(* PLC project Система умного дома.project, CODESYS CODESYS V3.5 SP17 Patch 3 *)
(* stored: creationDateTime 2026-04-06T20:38:17.5908527, modificationDateTime 2026-03-25T09:46:39.3897592 *)

{attribute 'qualified_only'}
{attribute 'strict'}
TYPE E_ALERT_PRIORITY : (ALERT_PRIORITY_NONE := 0, ALERT_PRIORITY_LOW := 1, ALERT_PRIORITY_MEDIUM := 2, ALERT_PRIORITY_HIGH := 3, ALERT_PRIORITY_CRITICAL := 4) BYTE;
END_TYPE

{attribute 'qualified_only'}
{attribute 'strict'}
TYPE E_Debug_Log_Level : (LOG_LEVEL_MINIMAL := 0, LOG_LEVEL_NORMAL := 1, LOG_LEVEL_VERBOSE := 2, LOG_LEVEL_DEBUG := 3) BYTE;
END_TYPE

{attribute 'qualified_only'}
{attribute 'strict'}
TYPE E_Lifetime_Device_Type : (LIFETIME_DEVICE_PUMP := 1, LIFETIME_DEVICE_FAN := 2) BYTE;
END_TYPE

{attribute 'qualified_only'}
{attribute 'strict'}
TYPE E_Outdoor_Mode : (OUTDOOR_MODE_AUTO := 0, OUTDOOR_MODE_PARTY := 1, OUTDOOR_MODE_SECURITY := 2, OUTDOOR_MODE_ECONOMY := 3, OUTDOOR_MODE_MANUAL := 4) BYTE;
END_TYPE

{attribute 'qualified_only'}
{attribute 'strict'}
TYPE E_PLC_ROLE : (ROLE_UNDEFINED := 0, ROLE_ACTIVE := 1, ROLE_STANDBY := 2, ROLE_OFFLINE := 3) USINT;
END_TYPE

{attribute 'qualified_only'}
{attribute 'strict'}
TYPE E_Rule_Action_Type : (ACTION_NONE := 0, ACTION_SET_FLOOR_HEATING := 1, ACTION_SET_LIGHTING_BASE := 2, ACTION_SET_LIGHTING_ACCENT := 3, ACTION_SET_SOCKET := 4, ACTION_SET_VENTILATION := 5, ACTION_SET_BLINDS := 6, ACTION_ACTIVATE_SCENARIO := 7, ACTION_TOGGLE_LIGHTING := 8, ACTION_TOGGLE_SOCKET := 9) BYTE;
END_TYPE

{attribute 'qualified_only'}
{attribute 'strict'}
TYPE E_Rule_Comparison : (COMP_NONE := 0, COMP_EQ := 1, COMP_GT := 2, COMP_LT := 3, COMP_GE := 4, COMP_LE := 5, COMP_IN_RANGE := 6, COMP_TRUE := 7, COMP_FALSE := 8) BYTE;
END_TYPE

(* values of E_Rule_Condition_Type: COND_AND: Логическое И (Rule Chaining); COND_OR: Логическое ИЛИ (Rule Chaining) *)

{attribute 'qualified_only'}
{attribute 'strict'}
TYPE E_Rule_Condition_Type : (COND_NONE := 0, COND_AIR_TEMP := 1, COND_FLOOR_TEMP := 2, COND_HUMIDITY := 3, COND_CO2 := 4, COND_METHANE := 5, COND_CO := 6, COND_DOOR_WINDOW := 7, COND_FLOOD := 8, COND_SMOKE := 9, COND_MOTION := 10, COND_TIME_OF_DAY := 11, COND_DAY_OF_WEEK := 12, COND_AND := 13, COND_OR := 14) BYTE;
END_TYPE

{attribute 'qualified_only'}
{attribute 'strict'}
TYPE E_SCENARIO_TYPE : (SCENARIO_NONE := 0, SCENARIO_MORNING := 1, SCENARIO_EVENING := 2, SCENARIO_AWAY := 3, SCENARIO_PARTY := 4, SCENARIO_SLEEP := 5, SCENARIO_EMERGENCY := 6, SCENARIO_PRESENCE := 7) BYTE;
END_TYPE

{attribute 'qualified_only'}
{attribute 'strict'}
TYPE E_SENSOR_TYPE : (SENSOR_TYPE_NONE := 0, SENSOR_TYPE_DOOR_WINDOW := 5, SENSOR_TYPE_GLASS_BREAK := 6, SENSOR_TYPE_FLOOD := 7, SENSOR_TYPE_SMOKE := 8, SENSOR_TYPE_GAS_METHANE := 1, SENSOR_TYPE_GAS_CO := 2, SENSOR_TYPE_TEMP_FLOOR := 3, SENSOR_TYPE_TEMP_AIR := 4) USINT;
END_TYPE

{attribute 'qualified_only'}
{attribute 'strict'}
TYPE E_Trend_Parameter_Type : (TREND_PARAM_NONE := 0, TREND_PARAM_TEMP_AIR := 1, TREND_PARAM_TEMP_FLOOR := 2, TREND_PARAM_PRESSURE := 3, TREND_PARAM_PUMP_CURRENT := 4, TREND_PARAM_GAS_METHANE := 5, TREND_PARAM_GAS_CO := 6) BYTE;
END_TYPE

{attribute 'qualified_only'}
{attribute 'strict'}
TYPE E_TwoFactor_Method : (TF_METHOD_NONE := 0, TF_METHOD_RFID := 1, TF_METHOD_TOTP := 2, TF_METHOD_BOTH := 3) BYTE;
END_TYPE

{attribute 'qualified_only'}
{attribute 'strict'}
TYPE E_Valve_Test_Result : (TEST_RESULT_NONE := 0, TEST_RESULT_PASSED := 1, TEST_RESULT_CURRENT_DEVIATION := 2, TEST_RESULT_TIME_DEVIATION := 3, TEST_RESULT_STALL := 4, TEST_RESULT_LIMIT_SWITCH_FAIL := 5, TEST_RESULT_ABORTED := 6) BYTE;
END_TYPE

(* values of E_VALVE_TYPE: VALVE_NC: Нормально-закрытый; VALVE_NO: Нормально-открытый *)

{attribute 'qualified_only'}
{attribute 'strict'}
TYPE E_VALVE_TYPE : (VALVE_NC := 1, VALVE_NO := 2) USINT;
END_TYPE

{attribute 'qualified_only'}
{attribute 'strict'}
TYPE E_VENTILATION_LOCATION : (VENT_LOCATION_NONE := 0, VENT_LOCATION_BASEMENT_GAME_ROOM := 1, VENT_LOCATION_BASEMENT_GYM := 2, VENT_LOCATION_BASEMENT_BOILER_ROOM := 3, VENT_LOCATION_BATHROOM_1F := 4, VENT_LOCATION_BATHROOM_2F := 5, VENT_LOCATION_MASTER_BATHROOM := 6, VENT_LOCATION_LAUNDRY := 7, VENT_LOCATION_KITCHEN := 8) BYTE;
END_TYPE

{attribute 'qualified_only'}
{attribute 'strict'}
TYPE E_VENTILATION_UNIT_TYPE : (VENTILATION_TYPE_NONE := 0, VENTILATION_TYPE_SUPPLY := 1, VENTILATION_TYPE_EXHAUST := 2) USINT;
END_TYPE

{attribute 'qualified_only'}
{attribute 'strict'}
TYPE E_WEATHER_COMPENSATION_METHOD : (WEATHER_COMP_NONE := 0, WEATHER_COMP_OUTDOOR_RESET := 1) USINT;
END_TYPE

{attribute 'qualified_only'}
{attribute 'strict'}
TYPE E_Zone_Access_Level : (ZONE_ACCESS_NONE := 0, ZONE_ACCESS_VIEW := 1, ZONE_ACCESS_CONTROL := 2, ZONE_ACCESS_CONFIG := 3, ZONE_ACCESS_FULL := 4) BYTE;
END_TYPE

TYPE ST_Astro_Time : STRUCT
  sunrise_ms : UDINT := 0;
  sunset_ms : UDINT := 0;
  is_daylight : BOOL := FALSE;
END_STRUCT;
END_TYPE

TYPE ST_BlackBox_Record : STRUCT
  Timestamp : UDINT;
  Gas_Methane_LEL : REAL;
  Gas_CO_PPM : REAL;
  Flood_Active : BOOL;
  Fire_Active : BOOL;
  Valve_Gas_Status : BYTE;
  Valve_Water_Status : BYTE;
  PLC_Active_ID : BYTE;
END_STRUCT;
END_TYPE

TYPE ST_Boiler_Status : STRUCT
  Active : BOOL;
  Running : BOOL;
  Error : BOOL;
  Power_Percent : REAL;
  Current_Power : REAL;
  Work_Seconds : UDINT;
  Work_Hours : REAL;
  Resource_Percent : REAL := 100;
  Last_Start : DT;
END_STRUCT;
END_TYPE

TYPE ST_Component_Maintenance : STRUCT
  Is_Faulty : BOOL;  (* Устройство неисправно *)
  Is_In_Maintenance : BOOL;  (* Выведено в ремонт вручную *)
  Fallback_Value : REAL;  (* Значение для подстановки (0-100% или температура) *)
  Use_Last_Good_Value : BOOL;  (* Использовать последнее достоверное значение *)
END_STRUCT;
END_TYPE

TYPE ST_Debug_Log_Record : STRUCT
  timestamp_ms : UDINT;
  level : BYTE;  (* E_Debug_Log_Level *)
  source_id : BYTE;
  event_code : WORD;
  value_int : UDINT;
  value_real : REAL;
  text : STRING(80);
  crc32 : DWORD;
END_STRUCT;
END_TYPE

TYPE ST_Debug_Logger_Config : STRUCT
  enabled : BOOL;
  sampling_period_ms : UDINT := 1000;
END_STRUCT;
END_TYPE

TYPE ST_Device_Health : STRUCT
  Health_Score : BYTE := 100;  (* 0..100% *)
  Total_Runtime_Hours : UDINT;
  Starts_Count : UDINT;
  Last_Start_Current : REAL;
  Avg_Start_Current : REAL;
  Maintenance_Required : BOOL;
  Warning_Message : STRING(50);
END_STRUCT;
END_TYPE

TYPE ST_DHW_Config : STRUCT
  Target_Temp : REAL := 55;
  Hysteresis : REAL := 2;
  Circulation_Schedule_Enabled : BOOL := TRUE;
  Circulation_Start : TOD := TIME_OF_DAY#6:0;
  Circulation_End : TOD := TIME_OF_DAY#23:0;
  Anti_Legionella_Enabled : BOOL := TRUE;
  Anti_Legionella_Day : UINT := 7;  (* Воскресенье *)
END_STRUCT;
END_TYPE

TYPE ST_DHW_Status : STRUCT
  Temp : REAL;
  Pressure : REAL;
  Heating_Pump_On : BOOL;
  Circ_Pump_On : BOOL;
  Error : BOOL;
  Error_ID : WORD;
END_STRUCT;
END_TYPE

TYPE ST_Flood_Config : STRUCT
  Emergency_Two_Stage_Enabled : BOOL := TRUE;  (* ТЗ 4.4 *)
  Valve_Test_Period_Days : UINT := 7;  (* ТЗ 12.2 *)
  Current_Threshold_MA : REAL := 500;  (* Порог тока для диагностики *)
END_STRUCT;
END_TYPE

TYPE ST_Flood_Global_Config : STRUCT
  valve_types : ARRAY[1..3] OF E_VALVE_TYPE := [3(E_VALVE_TYPE.VALVE_NC)];
  min_duration_ms : UDINT := 30000;
END_STRUCT;
END_TYPE

TYPE ST_FloorHeating_Circuit_Config : STRUCT
  circuit_id : BYTE := 0;
  zone : BYTE := 0;
  design_temp : REAL := 35;
  min_temp : REAL := 20;
  max_temp : REAL := 45;
  pid_kp : REAL := 2;
END_STRUCT;
END_TYPE

TYPE ST_FloorHeating_Global_Config : STRUCT
  enable_floor_heating : BOOL := TRUE;
  anti_freeze_temp : REAL := 7;
  overheat_temp : REAL := 45;
  weather_compensation_enabled : BOOL := TRUE;
  total_circuits : BYTE := 16;
END_STRUCT;
END_TYPE

TYPE ST_FloorHeating_Manifold_Config : STRUCT
  manifold_id : BYTE;
  location : STRING(30);
  nominal_flow : REAL;
  enable_pump : BOOL;
  circuits : ARRAY[1..4] OF ST_FloorHeating_Circuit_Config;
END_STRUCT;
END_TYPE

TYPE ST_Gas_Valve_Configuration : STRUCT
  valve_id : BYTE := 0;
  valve_type : E_VALVE_TYPE := E_VALVE_TYPE.VALVE_NC;
  close_time_seconds : UDINT := 10;
  open_time_seconds : UDINT := 10;
  emergency_open_allowed : BOOL := FALSE;
END_STRUCT;
END_TYPE

TYPE ST_Gateway_Command : STRUCT
  command_id : UDINT;
  timestamp_ms : UDINT;
  operator_id : STRING(10);
  command_type : BYTE;
  target_zone : BYTE;
  target_value : REAL;
  target_on_off : BOOL;
  target_scenario : E_SCENARIO_TYPE;
  target_armed : BOOL;
  crc32 : DWORD;
END_STRUCT;
END_TYPE

TYPE ST_Heating_Config : STRUCT
  Weather_Comp_Enabled : BOOL := TRUE;
  Weather_Coef : REAL := 0.1;
  Freeze_Threshold : REAL := 7;
  Overheat_Threshold : REAL := 45;
  Night_Reduction : REAL := 3;
  Target_Floor_Temp : REAL := 28;
  Target_Room_Temp : REAL := 22;
  Hysteresis : REAL := 0.5;
END_STRUCT;
END_TYPE

TYPE ST_History_Record : STRUCT
  timestamp_ms : UDINT := 0;
  event_code : WORD := 0;
  event_value : REAL := 0;
  unit : BYTE := 0;
  zone_id : BYTE := 0;
  operator_id : STRING(10) := '';
  priority : E_ALERT_PRIORITY := E_ALERT_PRIORITY.ALERT_PRIORITY_NONE;
END_STRUCT;
END_TYPE

TYPE ST_Lifetime_Status : STRUCT
  device_id : BYTE;
  runtime_hours : UDINT;
  start_count : UDINT;
  remaining_hours : UDINT;
  remaining_percent : BYTE;
  maintenance_required : BOOL;
  last_calc_timestamp : UDINT;
END_STRUCT;
END_TYPE

TYPE ST_Maintenance_Access_Config : STRUCT
  maintenance_enabled : BOOL := FALSE;
  max_duration_minutes : UDINT := 60;
  requires_two_person : BOOL := TRUE;
  access_level_required : BYTE := 2;
END_STRUCT;
END_TYPE

TYPE ST_Manifold_Status : STRUCT
  Pump_On : BOOL;
  Pump_Current : REAL;
  Pressure : REAL;
  Temp_Supply : REAL;
  Temp_Return : REAL;
  Valve_Pos : REAL;  (* 0-100% *)
  Error : BOOL;
  Error_ID : WORD;
END_STRUCT;
END_TYPE

TYPE ST_Operator_Zone_Rights : STRUCT
  operator_id : STRING(10);
  global_access_level : BYTE := 0;
  zone_masks : ARRAY[1..18] OF DWORD;
  last_modified : UDINT;
END_STRUCT;
END_TYPE

TYPE ST_Outdoor_Zone_Config : STRUCT
  zone_id : BYTE := 0;
  lighting_circuit_id : BYTE := 0;
  auto_enabled : BOOL := TRUE;
  party_mode_enabled : BOOL := FALSE;
END_STRUCT;
END_TYPE

TYPE ST_Owen_Analog_Value : STRUCT
  rValue : REAL;  (* Измеренное значение *)
  uiCycleTime : UINT;  (* Циклическое время *)
  wStatus : WORD;  (* Код статуса (ANALOG_SENSOR_ERRORS) *)
END_STRUCT;
END_TYPE

TYPE ST_Rule_Action : STRUCT
  Active : BOOL;
  Target_ID : BYTE;
  Value : REAL;
END_STRUCT;
END_TYPE

TYPE ST_Scenario_Config : STRUCT
  scenario_id : E_SCENARIO_TYPE;
  lighting_level_base : BYTE := 100;
  lighting_level_accent : BYTE := 100;
  floor_heating_adjust_celsius : REAL := 0;
  ventilation_speed_percent : BYTE := 50;
  sockets_enabled : BOOL := TRUE;
  blinds_position_percent : BYTE := 0;
END_STRUCT;
END_TYPE

TYPE ST_Scenario_Transition_Config : STRUCT
  current_scenario : E_SCENARIO_TYPE;
  target_scenario : E_SCENARIO_TYPE;
  min_duration_minutes : UDINT := 5;
  transition_allowed : BOOL := FALSE;
END_STRUCT;
END_TYPE

TYPE ST_Security_Config : STRUCT
  PIN_Code : STRING(4) := '1234';
  Max_Attempts : UINT := 3;
  Entry_Delay_S : UINT := 45;
  Two_Factor_Enabled : BOOL := FALSE;
  Two_Stage_Mode : BOOL := TRUE;  (* ТЗ 3.4 *)
  Confirmation_Timeout_S : UINT := 120;  (* ТЗ 3.4 (60-300с) *)
  Phones : ARRAY[1..5] OF STRING(15);
  gate_open_pulse_ms : UDINT := 1000;  (* Управление доступом *)
  wicket_open_pulse_ms : UDINT := 1000;
  lock_open_pulse_ms : UDINT := 1000;
  lock_close_pulse_ms : UDINT := 1000;
END_STRUCT;
END_TYPE

TYPE ST_Security_Global_Config : STRUCT
  entry_delay_seconds : UDINT := 30;
  exit_delay_seconds : UDINT := 60;
  alarm_duration_seconds : UDINT := 180;
  two_person_timeout_seconds : UDINT := 120;
  max_access_attempts : BYTE := 3;
  auto_arm_enabled : BOOL := FALSE;
  auto_arm_time_ms : UDINT := 0;
  gate_open_pulse_ms : UDINT := 1000;  (* ТЗ: Управление доступом *)
  wicket_open_pulse_ms : UDINT := 1000;
  lock_open_pulse_ms : UDINT := 1000;
  lock_close_pulse_ms : UDINT := 1000;
END_STRUCT;
END_TYPE

TYPE ST_Security_Zone_State : STRUCT
  Armed : BOOL;
  Alarm : BOOL;
  Bypassed : BOOL;
  Last_Trigger_Time : DT;
  Trigger_Count : UINT;
END_STRUCT;
END_TYPE

TYPE ST_Sensor_Calibration_Record : STRUCT
  sensor_id : UDINT := 0;
  sensor_type : E_SENSOR_TYPE;
  zone_id : BYTE := 0;
  offset : REAL := 0;
  multiplier : REAL := 1;
  last_calibration_timestamp : UDINT := 0;
  verification_passed : BOOL := FALSE;
END_STRUCT;
END_TYPE

TYPE ST_State_Snapshot : STRUCT
  timestamp_ms : UDINT := 0;
  operator_id : STRING(10) := '';
  scenario_id : E_SCENARIO_TYPE := E_SCENARIO_TYPE.SCENARIO_NONE;
  lighting_levels : ARRAY[1..16] OF BYTE;
  floor_heating_setpoints : ARRAY[1..16] OF REAL;
  alarm_active : BOOL := FALSE;
  crc32 : DWORD := 0;
END_STRUCT;
END_TYPE

TYPE ST_System_State_Summary : STRUCT
  Outdoor_Temp : REAL;
  Indoor_Temp : ARRAY[1..16] OF REAL;
  Floor_Temps : ARRAY[1..16] OF REAL;
  Humidity : ARRAY[1..8] OF REAL;
  CO2 : ARRAY[1..8] OF REAL;
  Gas_Alarm : BOOL;
  Flood_Alarm : BOOL;
  Fire_Alarm : BOOL;
  Security_Armed : BOOL;
END_STRUCT;
END_TYPE

TYPE ST_Tariff_Config : STRUCT
  Enabled : BOOL := FALSE;
  Night_Start_Hour : UINT := 23;  (* 23:00 *)
  Night_End_Hour : UINT := 7;  (* 07:00 *)
  Boost_Delta : REAL := 2;  (* На сколько градусов поднять уставку ночью *)
END_STRUCT;
END_TYPE

TYPE ST_Trend_Config : STRUCT
  param_type : BYTE;  (* E_Trend_Parameter_Type *)
  zone_id : BYTE;
  enabled : BOOL;
  deviation_threshold_percent : REAL := 10;
  history_days : UDINT := 7;
END_STRUCT;
END_TYPE

TYPE ST_Trend_Data : STRUCT
  config : ST_Trend_Config;
  record_count : UDINT;
  write_index : UDINT;
  sum_values : REAL;
  crc32 : DWORD;
END_STRUCT;
END_TYPE

TYPE ST_Trend_Header : STRUCT
  parameter_type : BYTE;  (* E_Trend_Parameter_Type *)
  zone_id : BYTE := 0;
  records_count : UDINT := 0;
  average_value : REAL := 0;
  min_value : REAL := 0;
  max_value : REAL := 0;
END_STRUCT;
END_TYPE

TYPE ST_Trend_History_Record : STRUCT
  timestamp_ms : UDINT := 0;
  value : REAL := 0;
END_STRUCT;
END_TYPE

TYPE ST_TwoFactor_Auth_State : STRUCT
  operator_id : STRING(10);
  is_pending : BOOL;  (* Ожидание ввода 2-го фактора *)
  start_time : UDINT;
  timeout_ms : UDINT := 60000;
END_STRUCT;
END_TYPE

TYPE ST_TwoFactor_Data : STRUCT
  operator_id : STRING(10);
  AuthMethod : BYTE;  (* E_TwoFactor_Method *)
  rfid_tag : STRING(20);
  totp_secret : STRING(32);
  last_modified : UDINT;
END_STRUCT;
END_TYPE

TYPE ST_User_Rule : STRUCT
  Enabled : BOOL;
  Condition_Type : BYTE;  (* 1-Temp, 2-Hum, 3-CO2, 4-Security, 5-Time *)
  Condition_Op : BYTE;  (* 1:>, 2:<, 3:= *)
  Condition_Value : REAL;
  Action_Target_ID : BYTE;
  Action_Value : REAL;
  Action_Type : BYTE;  (* 1-SetTemp, 2-Switch, 3-Scenario *)
  Priority : BYTE;  (* ТЗ 7.4: Приоритет (0-255) *)
END_STRUCT;
END_TYPE

TYPE ST_Valve_Test_Config : STRUCT
  valve_id : BYTE := 0;
  test_interval_days : UDINT := 7;
  nominal_current_a : REAL := 0.5;
  Nominal_Current : REAL := 0.5;
  nominal_close_time_sec : REAL := 10;
  enabled : BOOL := TRUE;
END_STRUCT;
END_TYPE

TYPE ST_Ventilation_Config : STRUCT
  CO2_Threshold : REAL := 800;
  Humidity_Threshold : REAL := 65;
  Night_Mode_Start : TOD := TIME_OF_DAY#23:0;
  Night_Mode_End : TOD := TIME_OF_DAY#7:0;
END_STRUCT;
END_TYPE

TYPE ST_Ventilation_Global_Config : STRUCT
  enable_ventilation : BOOL := TRUE;
  total_units : BYTE := 8;
  default_supply_speed : BYTE := 40;
  default_exhaust_speed : BYTE := 40;
END_STRUCT;
END_TYPE

TYPE ST_Ventilation_Scenario_Mode : STRUCT
  Scenario_ID : BYTE;
  Scenario_Priority : BYTE;
  Fire_Alarm : BOOL;
  Methane_Alarm : BOOL;
  Smoke_Detected : BOOL;
  Exhaust_Modes : ARRAY[1..5] OF BYTE;
  Supply_Modes : ARRAY[1..3] OF BYTE;
END_STRUCT;
END_TYPE

TYPE ST_Ventilation_Unit : STRUCT
  Enabled : BOOL;
  Speed_Percent : REAL;
  Filter_Dirty : BOOL;
  Error : BOOL;
  Mode : BYTE;  (* 0-Eco, 1-Std, 2-Int, 3-Emergency *)
END_STRUCT;
END_TYPE

TYPE ST_Ventilation_Unit_Config : STRUCT
  unit_id : BYTE := 0;
  unit_type : E_VENTILATION_UNIT_TYPE;
  location : E_VENTILATION_LOCATION;
  min_speed : BYTE := 20;
  max_speed : BYTE := 100;
  Threshold_Hum : REAL := 65;
  has_smoke_detector : BOOL := FALSE;
END_STRUCT;
END_TYPE

TYPE ST_Zone_Sensors : STRUCT
  Temp_Room : REAL;
  Temp_Floor : REAL;
  Motion_Active : BOOL;
  Switch_Physical : BOOL;
  Light_State : BOOL;
  Maintenance : ST_Component_Maintenance;
END_STRUCT;
END_TYPE

{attribute 'qualified_only'}
VAR_GLOBAL  (* GVL_BlackBox *)
  G_BlackBox_Buffer : ARRAY[0..99] OF ST_BlackBox_Record;  (* Буфер на 100 записей (при опросе 100мс это 10 секунд истории) *)
  G_BlackBox_Frozen : BOOL;
  G_BlackBox_LastIndex : INT;
END_VAR

{attribute 'qualified_only'}
VAR_GLOBAL CONSTANT  (* GVL_Constants *)
  C_MS_PER_SEC : UDINT := 1000;
  C_SEC_PER_MIN : UDINT := 60;
  C_MIN_PER_HOUR : UDINT := 60;
  C_MS_PER_MIN : UDINT := 60000;
  C_MAX_RULES : INT := 20;
  C_ZONE_COUNT : BYTE := 18;
END_VAR

{attribute 'qualified_only'}
VAR_GLOBAL  (* GVL_Diagnostics *)
  G_Pump_Health : ARRAY[1..5] OF ST_Device_Health;  (* Для 5 коллекторных насосов *)
  G_Gas_Valve_Health : ST_Device_Health;
  G_System_Health_Summary : BYTE := 100;
END_VAR

{attribute 'qualified_only'}
VAR_GLOBAL  (* GVL_Global_Variables *)
  GVL_System_Time_MS : UDINT;
  GVL_IsActivePLC : BOOL := TRUE;
  GVL_Local_PLC_Role : E_PLC_ROLE := E_PLC_ROLE.ROLE_ACTIVE;
  GVL_Floor_Temps : ARRAY[1..16] OF REAL;  (* Данные датчиков *)
  GVL_Valve_States : ARRAY[1..3] OF BYTE;
END_VAR

VAR_GLOBAL  (* GVL_HMI_Config *)
  G_HMI_FloorHeating_Configs : ARRAY[1..16] OF ST_FloorHeating_Circuit_Config;  (* Настройки отопления (16 контуров) *)
  G_HMI_Tariff_Settings : ST_Tariff_Config;
  G_HMI_Vent_Global_Config : ST_Ventilation_Global_Config;  (* Настройки вентиляции (8 установок) *)
  G_HMI_Vent_Unit_Configs : ARRAY[1..8] OF ST_Ventilation_Unit_Config;
  G_HMI_Scenario_Configs : ARRAY[1..6] OF ST_Scenario_Config;  (* Для каждого типа сценария *)
  G_HMI_Outdoor_Configs : ARRAY[1..4] OF ST_Outdoor_Zone_Config;
  G_HMI_Flood_Config : ST_Flood_Global_Config;  (* Настройки безопасности *)
  G_HMI_Cleaning_Mode_Active : ARRAY[1..3] OF BOOL;  (* Режим уборки для 3-х зон протечки *)
  G_HMI_Cleaning_Mode_TimeLeft : ARRAY[1..3] OF UINT;  (* Оставшееся время (мин) *)
  G_HMI_Gas_Config : ST_Gas_Valve_Configuration;
  G_HMI_Admin_2FA_Enabled : BOOL := FALSE;  (* Настройка: 1 или 2 фактора для ADMIN *)
  G_HMI_Current_Operator_Factor2_Done : BOOL;  (* Флаг прохождения 2-го фактора *)
  G_HMI_Sensor_Calibrations : ARRAY[1..20] OF ST_Sensor_Calibration_Record;  (* Калибровка датчиков (например, для 20 датчиков) *)
  G_HMI_Current_Operator_ID : STRING(10);  (* ID текущего авторизованного пользователя *)
  G_HMI_Manual_Gas_Valve_Open : BOOL;  (* Запрос на открытие *)
  G_HMI_Manual_Gas_Valve_Time : UDINT := 5;  (* Время в минутах *)
  G_HMI_Manual_Gas_Valve_TimeLeft : UDINT;  (* Оставшееся время (для вывода на HMI) *)
  G_HMI_Apply_Settings : BOOL;  (* Команда на сохранение настроек в NVRAM *)
  G_HMI_Gate_Open_Req : BOOL;  (* Управление доступом (HMI) *)
  G_HMI_Wicket_Open_Req : BOOL;
  G_HMI_Lock_1_Open_Req : BOOL;
  G_HMI_Lock_1_Close_Req : BOOL;
  G_HMI_Lock_2_Open_Req : BOOL;
  G_HMI_Lock_2_Close_Req : BOOL;
END_VAR

VAR_GLOBAL  (* GVL_IO *)
  DI_Security_Open : ARRAY[1..15] OF BOOL;  (* Датчики открытия (15 физических каналов по ТЗ 3.1) *)
  DI_Security_Glass : ARRAY[1..15] OF BOOL;  (* Датчики разбития (15 физических каналов по ТЗ 3.2) *)
  DI_Security_2F_Group : BOOL;  (* Групповой канал 2-го этажа *)
  DI_Flood_Sensors : ARRAY[1..12] OF BOOL;  (* Датчики протечки (12 штук по ТЗ 4.1) *)
  AO_Manifold_Valves : ARRAY[1..5] OF UINT;  (* 0-1000 (Modbus) *)
  DO_Manifold_Pumps : ARRAY[1..5] OF BOOL;
  AI_Manifold_Currents : ARRAY[1..5] OF INT;  (* 4-20mA -> 400-2000 *)
  AI_Manifold_Pressures : ARRAY[1..5] OF INT;  (* 0-10V -> 0-1000 *)
  AI_Manifold_Temps_Supply : ARRAY[1..5] OF ST_Owen_Analog_Value;
  AI_Manifold_Temps_Return : ARRAY[1..5] OF INT;
  AO_Supply_Fans : ARRAY[1..3] OF UINT;  (* 0-1000 *)
  AO_Exhaust_Fans : ARRAY[1..5] OF UINT;  (* 0-1000 *)
  DO_Boiler_Enable : ARRAY[1..2] OF BOOL;  (* Котлы (BAXI Luna Platinum+ через OpenTherm) *)
  AO_Boiler_Setpoint : ARRAY[1..2] OF UINT;  (* 0-1000 (0-100.0 C) *)
  AI_Boiler_Modulation : ARRAY[1..2] OF INT;
  AI_Boiler_Flame_Status : ARRAY[1..2] OF BOOL;
  DI_Boiler_Error : ARRAY[1..2] OF BOOL;
  AI_Methane_LEL : ARRAY[1..2] OF ST_Owen_Analog_Value;  (* 0-100% LEL *)
  AI_CO_PPM : ARRAY[1..8] OF REAL;  (* 0-1000 PPM *)
  DI_Smoke_Sensors : ARRAY[1..6] OF BOOL;
  AI_Temp_Outdoor : ST_Owen_Analog_Value;  (* Аналоговые входы (AI) *)
  AI_Floor_Temps : ARRAY[1..16] OF REAL;
  AI_Room_Temps : ARRAY[1..16] OF REAL;  (* Датчики температуры помещения (ТЗ 1.1) *)
  DO_Zone_Valves : ARRAY[1..16] OF BOOL;  (* Клапаны контуров ТП *)
  AI_DHW_Temp : REAL;  (* ГВС (ТЗ 5.0) *)
  AI_DHW_Pressure : REAL;
  DO_DHW_Heating_Pump : BOOL;
  DO_DHW_Circ_Pump : BOOL;
  DI_Lighting_Switches : ARRAY[1..16] OF BOOL;  (* Освещение и Движение (ТЗ 1.0, 2.0) *)
  DI_Motion_Sensors : ARRAY[1..16] OF BOOL;
  DO_Gas_Valve_Close : BOOL;  (* Безопасность и Аварии *)
  DO_Water_Valve_35_Close : BOOL;
  DO_Water_Valve_36_Close : BOOL;
  AI_Water_Valve_35_Current : REAL;
  AI_Water_Valve_36_Current : REAL;
  DI_Power_OK : BOOL;
  DO_Gas_Siren : BOOL;
  DO_Fire_Siren : BOOL;
  DO_Pump_Main_Enable : BOOL;
  DO_Gate_Open : BOOL;  (* Управление доступом (Сухие контакты) *)
  DO_Wicket_Open : BOOL;
  DO_Lock_1_Open : BOOL;
  DO_Lock_1_Close : BOOL;
  DO_Lock_2_Open : BOOL;
  DO_Lock_2_Close : BOOL;
END_VAR

VAR_GLOBAL  (* GVL_Vars *)
  G_System_Time_MS : UDINT;  (* Системное время (мс) *)
  G_Current_Scenario : E_SCENARIO_TYPE := E_SCENARIO_TYPE.SCENARIO_NONE;
  G_Security_Armed : BOOL := FALSE;
  G_Gas_Alarm_Active : BOOL := FALSE;
  G_Fire_Alarm_Active : BOOL := FALSE;
  G_Flood_Alarm_Active : BOOL := FALSE;
  G_Local_PLC_ID : BYTE := 1;  (* ID текущего ПЛК (1 для A, 2 для B) *)
  G_Active_PLC_ID : BYTE := 1;  (* ID активного ПЛК в данный момент *)
  G_Remote_PLC_Pulse : BOOL;  (* Импульс от партнера *)
  G_HMI_Current_Operator_ID : STRING(10) := 'ADMIN';  (* HMI и Конфигурация *)
  G_HMI_Gas_Config : ST_Gas_Valve_Configuration;
  G_Heating_Config : ST_Heating_Config;
  G_Ventilation_Config : ST_Ventilation_Config;
  G_DHW_Config : ST_DHW_Config;
  G_Security_Config : ST_Security_Config;
  G_Flood_Config : ST_Flood_Config;
  G_HMI_Mute_Alarm : BOOL;
  G_HMI_Manual_Gas_Valve_Open : BOOL;
  G_HMI_Manual_Gas_Valve_Time : UDINT := 300000;  (* 5 минут по умолчанию *)
  G_HMI_Manual_Gas_Valve_TimeLeft : UDINT;
  G_Floor_Temps : ARRAY[1..16] OF REAL;  (* Состояние датчиков *)
  G_BlackBox_Buffer : ARRAY[0..99] OF ST_BlackBox_Record;  (* Черный ящик *)
  G_BlackBox_LastIndex : INT;
  G_BlackBox_Frozen : BOOL;
  G_Maintenance_Zones : ARRAY[1..16] OF ST_Component_Maintenance;  (* ТЗ 6.0: Обслуживание и ремонт *)
  G_Maintenance_Manifolds : ARRAY[1..5] OF ST_Component_Maintenance;
  G_Maintenance_Lighting : ARRAY[1..16] OF ST_Component_Maintenance;
  G_HMI_Gate_Open_Req : BOOL;  (* Управление доступом (HMI) *)
  G_HMI_Wicket_Open_Req : BOOL;
  G_HMI_Lock_1_Open_Req : BOOL;
  G_HMI_Lock_1_Close_Req : BOOL;
  G_HMI_Lock_2_Open_Req : BOOL;
  G_HMI_Lock_2_Close_Req : BOOL;
END_VAR

INTERFACE IValveController
METHOD OpenValve : BOOL
  VAR_INPUT
    VI_Operator_ID : STRING(10);
    VI_Force : BOOL;
  END_VAR
END_METHOD
METHOD CloseValve : BOOL
  VAR_INPUT
    VI_Operator_ID : STRING(10);
    VI_Force : BOOL;
  END_VAR
END_METHOD
METHOD GetStatus : BYTE
END_METHOD
END_INTERFACE

PROGRAM PRG_PLC_A
  VAR
    L_PLC_ID : BYTE := 1;
  END_VAR

            // Установка глобального ID активного ПЛК (в реальной системе это определяется через механизм Heartbeat/Redundancy)
// Для ПЛК A: если он активен, G_Active_PLC_ID := 1
PRG_Main();

          
END_PROGRAM

PROGRAM PRG_PLC_B
  VAR
    L_PLC_ID : BYTE := 2;
  END_VAR

            // Для ПЛК B: если он активен, G_Active_PLC_ID := 2
PRG_Main();
          
END_PROGRAM

FUNCTION_BLOCK FB_Access_Control
  VAR_INPUT
    VI_System_Time_MS : UDINT;
    VI_IsActivePLC : BOOL;
    VI_Armed : BOOL;  (* Состояние охраны *)
    VI_Gate_Open_Req : BOOL;  (* Команды HMI *)
    VI_Wicket_Open_Req : BOOL;
    VI_Lock_1_Open_Req : BOOL;
    VI_Lock_1_Close_Req : BOOL;
    VI_Lock_2_Open_Req : BOOL;
    VI_Lock_2_Close_Req : BOOL;
    VI_Config : ST_Security_Config;  (* Настройки *)
  END_VAR
  VAR_OUTPUT
    VO_Gate_Open : BOOL;
    VO_Wicket_Open : BOOL;
    VO_Lock_1_Open : BOOL;
    VO_Lock_1_Close : BOOL;
    VO_Lock_2_Open : BOOL;
    VO_Lock_2_Close : BOOL;
  END_VAR
  VAR
    L_Gate_Timer : TON;
    L_Wicket_Timer : TON;
    L_Lock_1_Open_T : TON;
    L_Lock_1_Close_T : TON;
    L_Lock_2_Open_T : TON;
    L_Lock_2_Close_T : TON;
    L_Prev_Armed : BOOL;
    L_Auto_Lock_Req : BOOL;
  END_VAR

            IF NOT VI_IsActivePLC THEN
    RETURN;
END_IF;

// 1. Автоматическое закрытие при постановке на охрану
IF VI_Armed AND NOT L_Prev_Armed THEN
    L_Auto_Lock_Req := TRUE;
END_IF;
L_Prev_Armed := VI_Armed;

// 2. Логика импульсов
// Ворота
L_Gate_Timer(IN := VI_Gate_Open_Req, PT := TO_TIME(VI_Config.gate_open_pulse_ms));
VO_Gate_Open := VI_Gate_Open_Req AND NOT L_Gate_Timer.Q;

// Калитка
L_Wicket_Timer(IN := VI_Wicket_Open_Req, PT := TO_TIME(VI_Config.wicket_open_pulse_ms));
VO_Wicket_Open := VI_Wicket_Open_Req AND NOT L_Wicket_Timer.Q;

// Замок 1
L_Lock_1_Open_T(IN := VI_Lock_1_Open_Req, PT := TO_TIME(VI_Config.lock_open_pulse_ms));
VO_Lock_1_Open := VI_Lock_1_Open_Req AND NOT L_Lock_1_Open_T.Q;

L_Lock_1_Close_T(IN := (VI_Lock_1_Close_Req OR L_Auto_Lock_Req), PT := TO_TIME(VI_Config.lock_close_pulse_ms));
VO_Lock_1_Close := (VI_Lock_1_Close_Req OR L_Auto_Lock_Req) AND NOT L_Lock_1_Close_T.Q;

// Замок 2
L_Lock_2_Open_T(IN := VI_Lock_2_Open_Req, PT := TO_TIME(VI_Config.lock_open_pulse_ms));
VO_Lock_2_Open := VI_Lock_2_Open_Req AND NOT L_Lock_2_Open_T.Q;

L_Lock_2_Close_T(IN := (VI_Lock_2_Close_Req OR L_Auto_Lock_Req), PT := TO_TIME(VI_Config.lock_close_pulse_ms));
VO_Lock_2_Close := (VI_Lock_2_Close_Req OR L_Auto_Lock_Req) AND NOT L_Lock_2_Close_T.Q;

// Сброс авто-закрытия после завершения импульса
IF L_Lock_1_Close_T.Q AND L_Lock_2_Close_T.Q THEN
    L_Auto_Lock_Req := FALSE;
END_IF;

          
END_FUNCTION_BLOCK

FUNCTION_BLOCK FB_AccessCode_Manager
  VAR_INPUT
    VI_System_Time_MS : UDINT;
    VI_IsActivePLC : BOOL;
    VI_Code_To_Check : STRING(4);
  END_VAR
  VAR_OUTPUT
    VO_Code_Valid : BOOL;
  END_VAR
  VAR
    L_Codes : ARRAY[1..5] OF STRING(4) := ['1234', '5678', '0000', '1111', '2222'];
    L_i : INT;
  END_VAR

            VO_Code_Valid := FALSE;
FOR L_i := 1 TO 5 DO
    IF L_Codes[L_i] = VI_Code_To_Check THEN
        VO_Code_Valid := TRUE;
        RETURN;
    END_IF;
END_FOR;

          
END_FUNCTION_BLOCK

FUNCTION_BLOCK FB_Astro_Timer
  VAR_INPUT
    VI_System_Time_MS : UDINT;
    VI_Latitude : REAL := 55.75;  (* Москва *)
    VI_Longitude : REAL := 37.61;
  END_VAR
  VAR_OUTPUT
    VO_Sunset_Time : TOD;
    VO_Sunrise_Time : TOD;
    VO_Is_Night : BOOL;
  END_VAR
  VAR
    L_Current_TOD : TOD;
  END_VAR

            // Упрощенная логика астро-таймера (ТЗ 15.2)
// В реальном проекте используется библиотека SysTimeRtc или расчет по формулам
L_Current_TOD := UDINT_TO_TOD(VI_System_Time_MS MOD 86400000);

// Примерные значения для средней полосы
VO_Sunrise_Time := TOD#06:00;
VO_Sunset_Time := TOD#18:00;

// ТЗ 15.2: Закат + 30 мин / Рассвет - 30 мин
VO_Is_Night := (L_Current_TOD > (VO_Sunset_Time + T#30m)) OR (L_Current_TOD < (VO_Sunrise_Time - T#30m));

          
END_FUNCTION_BLOCK

FUNCTION_BLOCK FB_BlackBox_Recorder
  VAR_INPUT
    VI_Current_Data : ST_BlackBox_Record;
    VI_Freeze : BOOL;
  END_VAR
  VAR
    L_Write_Index : INT := 0;
    L_FileHandle : RTS_IEC_HANDLE;
    L_FileName : STRING := '/home/root/blackbox_dump.bin';
    L_FileResult : RTS_IEC_RESULT;
    L_State : INT;
  END_VAR

            CASE L_State OF
    0: // Циклическая запись
        IF NOT G_BlackBox_Frozen THEN
            G_BlackBox_Buffer[L_Write_Index] := VI_Current_Data;
            G_BlackBox_LastIndex := L_Write_Index;
            
            L_Write_Index := L_Write_Index + 1;
            IF L_Write_Index > 99 THEN
                L_Write_Index := 0;
            END_IF;
            
            IF VI_Freeze THEN
                G_BlackBox_Frozen := TRUE;
                L_State := 1;
            END_IF;
        END_IF;
        
    1: // Сохранение на Flash (SD-карту или внутреннюю память ПЛК210)
        L_FileHandle := SysFileOpen(L_FileName, AM_WRITE, ADR(L_FileResult));
        IF L_FileResult = 0 THEN
            SysFileWrite(L_FileHandle, ADR(G_BlackBox_Buffer[0]), SIZEOF(G_BlackBox_Buffer), ADR(L_FileResult));
            SysFileClose(L_FileHandle);
            L_State := 2;
        END_IF;
        
    2: // Завершено
        ;
END_CASE;

          
END_FUNCTION_BLOCK

FUNCTION_BLOCK FB_Boiler_Cascade_Controller
  VAR_INPUT
    VI_Demand_kW : REAL;
    VI_IsActivePLC : BOOL;
  END_VAR
  VAR_OUTPUT
    VO_Boiler1_On : BOOL;
    VO_Boiler2_On : BOOL;
  END_VAR
  VAR
    L_Lead_Boiler : BYTE := 1;  (* 1 или 2 *)
    L_Boiler1_Hours : UDINT;
    L_Boiler2_Hours : UDINT;
    L_Last_Hour_Update : UDINT;
    L_System_Time : UDINT;
  END_VAR
  VAR_INPUT
    VI_System_Time : UDINT;
  END_VAR

            // Логика ротации по наработке
IF (VI_System_Time - L_Last_Hour_Update) >= 3600000 THEN // Раз в час
    L_Last_Hour_Update := VI_System_Time;
    IF VO_Boiler1_On THEN L_Boiler1_Hours := L_Boiler1_Hours + 1; END_IF;
    IF VO_Boiler2_On THEN L_Boiler2_Hours := L_Boiler2_Hours + 1; END_IF;
    
    // Смена ведущего, если разница более 100 часов
    IF (L_Boiler1_Hours > L_Boiler2_Hours + 100) THEN
        L_Lead_Boiler := 2;
    ELSIF (L_Boiler2_Hours > L_Boiler1_Hours + 100) THEN
        L_Lead_Boiler := 1;
    END_IF;
END_IF;

IF VI_IsActivePLC THEN
    IF VI_Demand_kW > 24.0 THEN
        VO_Boiler1_On := TRUE;
        VO_Boiler2_On := TRUE;
    ELSIF VI_Demand_kW > 2.0 THEN
        VO_Boiler1_On := (L_Lead_Boiler = 1);
        VO_Boiler2_On := (L_Lead_Boiler = 2);
    ELSE
        VO_Boiler1_On := FALSE;
        VO_Boiler2_On := FALSE;
    END_IF;
END_IF;

          
END_FUNCTION_BLOCK

FUNCTION_BLOCK FB_Boiler_Cascade_Manager
  VAR_INPUT
    VI_Boiler1_Status : ST_Boiler_Status;
    VI_Boiler2_Status : ST_Boiler_Status;
    VI_Role_Swap_Interval : UDINT := 168;  (* часы *)
  END_VAR
  VAR_OUTPUT
    VO_Boiler1_Enable : BOOL;
    VO_Boiler2_Enable : BOOL;
  END_VAR

            // Логика п. 2.8: Включение резервного при >80% мощности или отказе
IF VI_Boiler1_Status.Error OR VI_Boiler1_Status.Current_Power > 80.0 THEN
    VO_Boiler2_Enable := TRUE;
ELSE
    VO_Boiler2_Enable := FALSE;
END_IF;

VO_Boiler1_Enable := NOT VI_Boiler1_Status.Error;

          
END_FUNCTION_BLOCK

FUNCTION_BLOCK FB_Calibration_Manager
  VAR_INPUT
    VI_Raw_Value : REAL;
    VI_Type : BYTE;  (* 1-Temp, 2-Pressure, 3-Gas *)
    VI_Calib_Record : ST_Sensor_Calibration_Record;
    VI_System_Time_MS : UDINT;
    VI_Start_Verification : BOOL;
  END_VAR
  VAR_OUTPUT
    VO_Calibrated_Value : REAL;
    VO_Verification_Active : BOOL;
    VO_Verification_Failed : BOOL;
    VO_Deviation_Percent : REAL;
  END_VAR
  VAR
    L_Verification_Timer : TON;
    L_Initial_Value : REAL;
  END_VAR

            // 1. Расчет калиброванного значения
CASE VI_Type OF
    1: VO_Calibrated_Value := VI_Raw_Value + VI_Calib_Record.offset;
    2, 3: VO_Calibrated_Value := (VI_Raw_Value * VI_Calib_Record.multiplier) + VI_Calib_Record.offset;
END_CASE;

// 2. Верификация через 1 час (ТЗ 9.5)
IF VI_Start_Verification AND NOT VO_Verification_Active THEN
    VO_Verification_Active := TRUE;
    L_Initial_Value := VO_Calibrated_Value;
    L_Verification_Timer(IN := TRUE, PT := T#1h);
END_IF;

L_Verification_Timer(IN := VO_Verification_Active);

IF L_Verification_Timer.Q THEN
    VO_Verification_Active := FALSE;
    L_Verification_Timer(IN := FALSE);
    
    // ТЗ 9.5: Отклонение ≤2.0% (норма) / >5.0% (ошибка)
    IF L_Initial_Value <> 0 THEN
        VO_Deviation_Percent := ABS(VO_Calibrated_Value - L_Initial_Value) / L_Initial_Value * 100.0;
    ELSE
        VO_Deviation_Percent := 0.0;
    END_IF;
    
    VO_Verification_Failed := (VO_Deviation_Percent > 5.0);
END_IF;

          
END_FUNCTION_BLOCK

FUNCTION_BLOCK FB_CO_Detector
  VAR_INPUT
    VI_CO_PPM : REAL;
    VI_Threshold_Warning : REAL := 30;
    VI_Threshold_Alarm : REAL := 70;
  END_VAR
  VAR_OUTPUT
    VO_Warning_Active : BOOL;
    VO_Alarm_Active : BOOL;
  END_VAR

            VO_Warning_Active := (VI_CO_PPM >= VI_Threshold_Warning);
VO_Alarm_Active := (VI_CO_PPM >= VI_Threshold_Alarm);

          
END_FUNCTION_BLOCK

FUNCTION_BLOCK FB_CRC32_Calculator
  VAR
    L_Table : ARRAY[0..255] OF DWORD;
    L_Initialized : BOOL := FALSE;
    L_i : INT;
    L_j : INT;
    L_Entry : DWORD;
  END_VAR

            
          

METHOD InitTable
                  IF L_Initialized THEN RETURN; END_IF;

FOR L_i := 0 TO 255 DO
    L_Entry := TO_DWORD(L_i);
    FOR L_j := 0 TO 7 DO
        IF (L_Entry AND 1) <> 0 THEN
            L_Entry := SHR(L_Entry, 1) XOR 16#EDB88320;
        ELSE
            L_Entry := SHR(L_Entry, 1);
        END_IF;
    END_FOR;
    L_Table[L_i] := L_Entry;
END_FOR;
L_Initialized := TRUE;
                
END_METHOD

METHOD Calculate : DWORD
  VAR_INPUT
    VI_DataPtr : POINTER TO BYTE;
    VI_Size : UDINT;
  END_VAR
  VAR
    L_k : UDINT;
    L_CRC : DWORD := 16#FFFFFFFF;
  END_VAR
                  InitTable();

IF VI_DataPtr = 0 OR VI_Size = 0 THEN
    Calculate := 0;
    RETURN;
END_IF;

FOR L_k := 0 TO VI_Size - 1 DO
    L_CRC := L_Table[TO_INT((L_CRC XOR VI_DataPtr[TO_INT(L_k)]) AND 16#FF)] XOR SHR(L_CRC, 8);
END_FOR;

Calculate := L_CRC XOR 16#FFFFFFFF;
                
END_METHOD
END_FUNCTION_BLOCK

FUNCTION_BLOCK FB_Debug_Logger
  VAR_INPUT
    VI_Config : ST_Debug_Logger_Config;
    VI_System_Time_MS : UDINT;
    VI_Floor_Temps : ARRAY[1..16] OF REAL;
    VI_Pump_Currents : ARRAY[1..5] OF REAL;
    VI_Error_Code : UDINT;
  END_VAR
  VAR
    L_buffer : ARRAY[1..1000] OF ST_Debug_Log_Record;
    L_write_idx : INT := 1;
    L_last_log_time : UDINT;
    L_i : INT;
  END_VAR

            // Цикл логирования
IF VI_Config.enabled AND (VI_System_Time_MS - L_last_log_time >= VI_Config.sampling_period_ms) THEN
    L_last_log_time := VI_System_Time_MS;
    
    // Логируем температуры (если изменились или по таймауту)
    FOR L_i := 1 TO 16 DO
        L_buffer[L_write_idx].timestamp_ms := VI_System_Time_MS;
        L_buffer[L_write_idx].level := E_Debug_Log_Level.LOG_LEVEL_VERBOSE;
        L_buffer[L_write_idx].source_id := TO_BYTE(L_i);
        L_buffer[L_write_idx].value_real := VI_Floor_Temps[L_i];
        L_buffer[L_write_idx].text := 'Floor Temp Update';
        
        L_write_idx := (L_write_idx MOD 1000) + 1;
    END_FOR;

    // Логируем ошибки
    IF VI_Error_Code <> 0 THEN
        L_buffer[L_write_idx].timestamp_ms := VI_System_Time_MS;
        L_buffer[L_write_idx].level := E_Debug_Log_Level.LOG_LEVEL_MINIMAL;
        L_buffer[L_write_idx].event_code := TO_WORD(VI_Error_Code);
        L_buffer[L_write_idx].text := 'System Error Detected';
        L_write_idx := (L_write_idx MOD 1000) + 1;
    END_IF;
END_IF;

          
END_FUNCTION_BLOCK

FUNCTION_BLOCK FB_Device_Predictive_Diag
  VAR_INPUT
    VI_Current_Value : REAL;  (* Текущий ток или время *)
    VI_Nominal_Value : REAL;  (* Эталонное значение *)
    VI_Is_Running : BOOL;
    VI_Reset_Stats : BOOL;
  END_VAR
  VAR_IN_OUT
    VIO_Health_Data : ST_Device_Health;
  END_VAR
  VAR
    L_Prev_Running : BOOL;
    L_Current_Sum : REAL;
    L_Sample_Count : UDINT;
  END_VAR

            // 1. Счётчик пусков и замер пускового тока
IF VI_Is_Running AND NOT L_Prev_Running THEN
    VIO_Health_Data.Starts_Count := VIO_Health_Data.Starts_Count + 1;
    VIO_Health_Data.Last_Start_Current := VI_Current_Value;
    
    // Обновление среднего пускового тока
    L_Sample_Count := L_Sample_Count + 1;
    L_Current_Sum := L_Current_Sum + VI_Current_Value;
    VIO_Health_Data.Avg_Start_Current := L_Current_Sum / UDINT_TO_REAL(L_Sample_Count);
END_IF;

// 2. Анализ отклонения (п. 12.1 ТЗ)
IF VI_Is_Running THEN
    // Если ток выше номинала на 50% - снижаем здоровье
    IF VI_Current_Value > (VI_Nominal_Value * 1.5) THEN
        IF VIO_Health_Data.Health_Score > 0 THEN
            VIO_Health_Data.Health_Score := VIO_Health_Data.Health_Score - 1;
        END_IF;
    END_IF;
END_IF;

// 3. Генерация предупреждения
IF VIO_Health_Data.Health_Score < 20 THEN
    VIO_Health_Data.Maintenance_Required := TRUE;
    VIO_Health_Data.Warning_Message := 'Критический износ: проверьте механику';
ELSIF VIO_Health_Data.Health_Score < 60 THEN
    VIO_Health_Data.Warning_Message := 'Предупреждение: повышенное трение';
END_IF;

L_Prev_Running := VI_Is_Running;

          
END_FUNCTION_BLOCK

FUNCTION_BLOCK FB_DHW_Manager
  VAR_INPUT
    VI_System_Time_MS : UDINT;
    VI_IsActivePLC : BOOL;
    VI_Temp : REAL;
    VI_Pressure : REAL;
    VI_Config : ST_DHW_Config;
    VI_Maintenance : ST_Component_Maintenance;
  END_VAR
  VAR_OUTPUT
    VO_Status : ST_DHW_Status;
    VO_Heating_Pump : BOOL;
    VO_Circ_Pump : BOOL;
  END_VAR
  VAR
    L_Current_TOD : TOD;
    L_Legionella_Active : BOOL;
    L_Last_Good_Temp : REAL := 55;
  END_VAR

            // 1. Обработка неисправности (ТЗ 7.0)
IF VI_Maintenance.Is_Faulty OR VI_Maintenance.Is_In_Maintenance THEN
    VO_Status.Temp := SEL(VI_Maintenance.Use_Last_Good_Value, VI_Maintenance.Fallback_Value, L_Last_Good_Temp);
ELSE
    VO_Status.Temp := VI_Temp;
    L_Last_Good_Temp := VI_Temp;
END_IF;

VO_Status.Pressure := VI_Pressure;

// 2. Логика нагрева
IF VI_IsActivePLC THEN
    IF VO_Status.Temp < (VI_Config.Target_Temp - VI_Config.Hysteresis) THEN
        VO_Heating_Pump := TRUE;
    ELSIF VO_Status.Temp > (VI_Config.Target_Temp + VI_Config.Hysteresis) THEN
        VO_Heating_Pump := FALSE;
    END_IF;
    
    // 3. Циркуляция ГВС по расписанию
    L_Current_TOD := UDINT_TO_TOD(VI_System_Time_MS MOD 86400000);
    VO_Circ_Pump := VI_Config.Circulation_Schedule_Enabled AND 
                    (L_Current_TOD >= VI_Config.Circulation_Start AND L_Current_TOD <= VI_Config.Circulation_End);
ELSE
    VO_Heating_Pump := FALSE;
    VO_Circ_Pump := FALSE;
END_IF;

VO_Status.Heating_Pump_On := VO_Heating_Pump;
VO_Status.Circ_Pump_On := VO_Circ_Pump;
VO_Status.Error := (VI_Pressure < 1.0 OR VI_Pressure > 4.0);

          
END_FUNCTION_BLOCK

FUNCTION_BLOCK FB_Emergency_Valve_Open
  VAR_INPUT
    VI_Fire_Alarm : BOOL;
    VI_Gas_Alarm : BOOL;
  END_VAR
  VAR_OUTPUT
    VO_Open_Cmd : BOOL;
  END_VAR

            // Приоритетное открытие при любой серьезной аварии
VO_Open_Cmd := VI_Fire_Alarm OR VI_Gas_Alarm;

          
END_FUNCTION_BLOCK

FUNCTION_BLOCK FB_Exhaust_Ventilation_Controller
  VAR_INPUT
    VI_Humidity : REAL;
    VI_CO2 : REAL;
    VI_Config : ST_Ventilation_Unit_Config;
  END_VAR
  VAR_OUTPUT
    VO_Fan_Speed : BYTE;
  END_VAR

            IF VI_Humidity > VI_Config.Threshold_Hum THEN
    VO_Fan_Speed := 100;
ELSIF VI_CO2 > 800.0 THEN
    VO_Fan_Speed := 70;
ELSE
    VO_Fan_Speed := 40;
END_IF;

          
END_FUNCTION_BLOCK

FUNCTION_BLOCK FB_Flood_Detector
  VAR_INPUT
    VI_Sensors : ARRAY[1..12] OF BOOL;
    VI_IsActivePLC : BOOL;
  END_VAR
  VAR_OUTPUT
    VO_Flood_Alarm : BOOL;
    VO_Close_Valve_35 : BOOL;
    VO_Close_Valve_36 : BOOL;
  END_VAR
  VAR
    L_i : INT;
  END_VAR

            VO_Flood_Alarm := FALSE;
VO_Close_Valve_35 := FALSE;
VO_Close_Valve_36 := FALSE;

FOR L_i := 1 TO 12 DO
    IF VI_Sensors[L_i] THEN
        VO_Flood_Alarm := TRUE;
        IF VI_IsActivePLC THEN
            // Логика п. 4.2: Зона 2 (4-5) и Зона 3 (6-7) делят клапан 36
            IF L_i >= 4 AND L_i <= 7 THEN
                VO_Close_Valve_36 := TRUE;
            ELSIF L_i >= 1 AND L_i <= 3 THEN
                VO_Close_Valve_35 := TRUE;
            END_IF;
        END_IF;
    END_IF;
END_FOR;

          
END_FUNCTION_BLOCK

FUNCTION_BLOCK FB_FloorHeating_Controller
  VAR_INPUT
    VI_Current_Temp : REAL;
    VI_Config : ST_FloorHeating_Circuit_Config;
    VI_Tariff : ST_Tariff_Config;
    VI_Current_Hour : UINT;
    VI_IsActivePLC : BOOL;
  END_VAR
  VAR_OUTPUT
    VO_Pump_Run : BOOL;
    VO_Valve_Pos : REAL;  (* 0..10V *)
    VO_Effective_Setpoint : REAL;
  END_VAR
  VAR
    L_Is_Night : BOOL;
  END_VAR

            // 1. Определение активного тарифа
IF VI_Tariff.Enabled THEN
    IF VI_Tariff.Night_Start_Hour > VI_Tariff.Night_End_Hour THEN
        // Переход через полночь (например, 23:00 - 07:00)
        L_Is_Night := (VI_Current_Hour >= VI_Tariff.Night_Start_Hour) OR (VI_Current_Hour < VI_Tariff.Night_End_Hour);
    ELSE
        // В пределах одного дня
        L_Is_Night := (VI_Current_Hour >= VI_Tariff.Night_Start_Hour) AND (VI_Current_Hour < VI_Tariff.Night_End_Hour);
    END_IF;
ELSE
    L_Is_Night := FALSE;
END_IF;

// 2. Расчет эффективной уставки
VO_Effective_Setpoint := VI_Config.design_temp;
IF L_Is_Night THEN
    VO_Effective_Setpoint := VO_Effective_Setpoint + VI_Tariff.Boost_Delta;
END_IF;

// 3. Простая логика управления (гистерезис)
IF VI_IsActivePLC THEN
    IF VI_Current_Temp < (VO_Effective_Setpoint - 0.5) THEN
        VO_Pump_Run := TRUE;
        VO_Valve_Pos := 10.0;
    ELSIF VI_Current_Temp > (VO_Effective_Setpoint + 0.5) THEN
        VO_Pump_Run := FALSE;
        VO_Valve_Pos := 0.0;
    END_IF;
END_IF;

          
END_FUNCTION_BLOCK

FUNCTION_BLOCK FB_FloorHeating_Freeze_Protection
  VAR_INPUT
    VI_Floor_Temps : ARRAY[1..16] OF REAL;
    VI_Outdoor_Temp : REAL;
    VI_Threshold : REAL := 7;
  END_VAR
  VAR_OUTPUT
    VO_Freeze_Alert : BOOL;
    VO_Pump_Force_On : BOOL;
  END_VAR
  VAR
    L_i : INT;
  END_VAR

            VO_Freeze_Alert := FALSE;
VO_Pump_Force_On := FALSE;

FOR L_i := 1 TO 16 DO
    IF VI_Floor_Temps[L_i] < VI_Threshold THEN
        VO_Freeze_Alert := TRUE;
        VO_Pump_Force_On := TRUE;
        RETURN;
    END_IF;
END_FOR;

IF VI_Outdoor_Temp < -5.0 THEN
    VO_Pump_Force_On := TRUE;
END_IF;

          
END_FUNCTION_BLOCK

FUNCTION_BLOCK FB_FloorHeating_Overheat_Protection
  VAR_INPUT
    VI_Temps : ARRAY[1..16] OF REAL;
    VI_Threshold : REAL := 45;
  END_VAR
  VAR_OUTPUT
    VO_Overheat_Detected : BOOL;
    VO_Locked_Circuits : ARRAY[1..16] OF BOOL;
  END_VAR
  VAR
    L_i : INT;
  END_VAR

            VO_Overheat_Detected := FALSE;
FOR L_i := 1 TO 16 DO
    IF VI_Temps[L_i] > VI_Threshold THEN
        VO_Overheat_Detected := TRUE;
        VO_Locked_Circuits[L_i] := TRUE;
    END_IF;
END_FOR;

          
END_FUNCTION_BLOCK

FUNCTION_BLOCK FB_Gas_Methane_Detector
  VAR_INPUT
    VI_Methane_LEL : REAL;
    VI_Threshold_Alarm : REAL := 20;
  END_VAR
  VAR_OUTPUT
    VO_Alarm_Active : BOOL;
    VO_Close_Valve : BOOL;
  END_VAR

            VO_Alarm_Active := (VI_Methane_LEL >= VI_Threshold_Alarm);
VO_Close_Valve := VO_Alarm_Active;

          
END_FUNCTION_BLOCK

FUNCTION_BLOCK FB_Gas_Smoke_Manager
  VAR_INPUT
    VI_System_Time_MS : UDINT;
    VI_IsActivePLC : BOOL;
    VI_Methane_LEL : ARRAY[1..2] OF REAL;
    VI_CO_PPM : ARRAY[1..8] OF REAL;
    VI_Smoke_Sensors : ARRAY[1..6] OF BOOL;
    VI_Mute_Request : BOOL;
  END_VAR
  VAR_OUTPUT
    VO_Gas_Alarm : BOOL;
    VO_Fire_Alarm : BOOL;
    VO_Siren_Active : BOOL;
    VO_Gas_Valve_Close : BOOL;
    VO_Boiler_Stop : BOOL;
    VO_Vent_PV3_Boost : BOOL;  (* ТЗ 5.1 (ПВ-3 при 10% LEL) *)
    VO_Supply_100_Req : BOOL;  (* ТЗ 6.4 (Метан >20%) *)
    VO_Exhaust_100_Req : BOOL;  (* ТЗ 6.4 (Пожар) *)
    VO_Supply_80_Req : BOOL;  (* ТЗ 5.4 (CO) *)
    VO_Status_Msg : STRING(200);
  END_VAR
  VAR
    L_Methane_Max : REAL;
    L_CO_Max : REAL;
    L_Smoke_Active : BOOL;
    L_Smoke_Timer : ARRAY[1..6] OF TON;
    L_Mute_Timer : TON;
    L_Muted : BOOL;
    L_Mute_Count : UINT;  (* ТЗ 5.5 *)
    L_i : INT;
    L_j : INT;
    L_Smoke_Count : UINT;
    L_CO_Timer_30ppm : TON;  (* 8 часов *)
    L_CO_Timer_70ppm : TON;  (* 1 час *)
    L_CO_Timer_400ppm : TON;  (* 15 минут *)
  END_VAR

            // 1. Обработка метана (ТЗ 5.1, 6.4)
L_Methane_Max := 0.0;
FOR L_i := 1 TO 2 DO IF VI_Methane_LEL[L_i] > L_Methane_Max THEN L_Methane_Max := VI_Methane_LEL[L_i]; END_IF; END_FOR;

VO_Vent_PV3_Boost := (L_Methane_Max >= 10.0); // ТЗ 5.1: ПВ-3 при 10% LEL

IF L_Methane_Max >= 40.0 THEN
    VO_Gas_Alarm := TRUE; VO_Gas_Valve_Close := TRUE; VO_Boiler_Stop := TRUE; VO_Supply_100_Req := TRUE;
    VO_Status_Msg := 'КРИТИЧЕСКАЯ УТЕЧКА ГАЗА (40% LEL)';
ELSIF L_Methane_Max >= 20.0 THEN
    VO_Gas_Alarm := TRUE; VO_Gas_Valve_Close := TRUE; VO_Boiler_Stop := TRUE; VO_Supply_100_Req := TRUE;
    VO_Status_Msg := 'УТЕЧКА ГАЗА (20% LEL)';
ELSIF L_Methane_Max >= 10.0 THEN 
    VO_Status_Msg := 'ПРЕДУПРЕЖДЕНИЕ: ГАЗ (10% LEL)';
END_IF;

// 2. Обработка CO (ТЗ 5.2, 5.4)
L_CO_Max := 0.0;
FOR L_i := 1 TO 8 DO IF VI_CO_PPM[L_i] > L_CO_Max THEN L_CO_Max := VI_CO_PPM[L_i]; END_IF; END_FOR;

L_CO_Timer_30ppm(IN := (L_CO_Max >= 30.0), PT := T#8h);
L_CO_Timer_70ppm(IN := (L_CO_Max >= 70.0), PT := T#1h);
L_CO_Timer_400ppm(IN := (L_CO_Max >= 400.0), PT := T#15m);

IF L_CO_Timer_400ppm.Q THEN VO_Gas_Alarm := TRUE; VO_Status_Msg := 'КРИТИЧЕСКАЯ КОНЦЕНТРАЦИЯ CO (400 ppm / 15 мин)';
ELSIF L_CO_Timer_70ppm.Q THEN VO_Gas_Alarm := TRUE; VO_Status_Msg := 'ВЫСОКАЯ КОНЦЕНТРАЦИЯ CO (70 ppm / 1 час)';
ELSIF L_CO_Timer_30ppm.Q THEN VO_Gas_Alarm := TRUE; VO_Status_Msg := 'ПОВЫШЕННАЯ КОНЦЕНТРАЦИЯ CO (30 ppm / 8 час)';
END_IF;

IF VO_Gas_Alarm AND L_CO_Max >= 30.0 THEN VO_Supply_80_Req := TRUE; END_IF; // ТЗ 5.4

// 3. Обработка дыма (ТЗ 5.3, 6.4)
L_Smoke_Count := 0;
FOR L_i := 1 TO 6 DO
    L_Smoke_Timer[L_i](IN := VI_Smoke_Sensors[L_i], PT := T#30s);
    IF VI_Smoke_Sensors[L_i] THEN L_Smoke_Count := L_Smoke_Count + 1; END_IF;
    // ТЗ 5.3: Верификация вторым датчиком ИЛИ сигнал > 30 сек
    IF L_Smoke_Timer[L_i].Q OR (L_Smoke_Count >= 2) THEN L_Smoke_Active := TRUE; END_IF;
END_FOR;

IF L_Smoke_Active THEN 
    VO_Fire_Alarm := TRUE; VO_Boiler_Stop := TRUE; VO_Exhaust_100_Req := TRUE;
    VO_Status_Msg := 'ПОЖАРНАЯ ТРЕВОГА: ДЫМ'; 
END_IF;

// 4. Сирена и квитирование (ТЗ 5.5)
IF VO_Gas_Alarm OR VO_Fire_Alarm THEN
    IF VI_Mute_Request AND NOT L_Muted AND L_Mute_Count < 3 THEN
        L_Muted := TRUE; L_Mute_Count := L_Mute_Count + 1;
        L_Mute_Timer(IN := TRUE, PT := T#5m);
    END_IF;
    
    L_Mute_Timer(IN := L_Muted);
    IF L_Mute_Timer.Q THEN L_Muted := FALSE; L_Mute_Timer(IN := FALSE); END_IF;
    VO_Siren_Active := NOT L_Muted;
ELSE
    L_Muted := FALSE; L_Mute_Count := 0; VO_Siren_Active := FALSE;
END_IF;

          
END_FUNCTION_BLOCK

FUNCTION_BLOCK FB_Gas_Valve_Controller IMPLEMENTS IValveController
  VAR_INPUT
    VI_System_Time : UDINT;
    VI_IsActivePLC : BOOL;
    VI_Gas_Alarm : BOOL;
    VI_Config : ST_Gas_Valve_Configuration;
  END_VAR
  VAR_OUTPUT
    VO_Valve_Closed : BOOL;
    VO_Status_Msg : STRING(200);
  END_VAR

            // При аварии газа - немедленное закрытие
IF VI_Gas_Alarm AND VI_IsActivePLC THEN
    VO_Valve_Closed := TRUE;
    VO_Status_Msg := 'ГАЗОВЫЙ КЛАПАН ЗАКРЫТ ПО АВАРИИ';
END_IF;
          

METHOD CloseValve : BOOL
  VAR_INPUT
    VI_Operator_ID : STRING(10);
    VI_Force : BOOL;
  END_VAR
                  VO_Valve_Closed := TRUE;
CloseValve := TRUE;
                
END_METHOD

METHOD GetStatus : BYTE
                  GetStatus := TO_BYTE(SEL(VO_Valve_Closed, 0, 1));
                
END_METHOD

METHOD OpenValve : BOOL
  VAR_INPUT
    VI_Operator_ID : STRING(10);
    VI_Force : BOOL;
  END_VAR
                  IF VI_IsActivePLC OR VI_Force THEN
    VO_Valve_Closed := FALSE;
    OpenValve := TRUE;
END_IF;
                
END_METHOD
END_FUNCTION_BLOCK

FUNCTION_BLOCK FB_Gateway_Interface
  VAR_INPUT
    VI_System_Time_MS : UDINT;
    VI_Local_PLC_Role : E_PLC_ROLE;
    VI_Incoming_Command : ST_Gateway_Command;
    VI_Command_Received : BOOL;
    VI_FloorHeating_Temps : ARRAY[1..16] OF REAL;  (* Состояния системы *)
    VI_Room_Temps : ARRAY[1..16] OF REAL;
    VI_Zone_Valve_States : ARRAY[1..16] OF BOOL;
    VI_Manifold_Pressures : ARRAY[1..5] OF REAL;
    VI_Manifold_Pump_States : ARRAY[1..5] OF BOOL;
    VI_Outdoor_Temp : REAL;
    VI_Security_Armed : BOOL;
    VI_Flood_Alarm_Active : BOOL;
    VI_Gas_Alarm_Active : BOOL;
    VI_Fire_Alarm_Active : BOOL;
    VI_Methane_Concentration : REAL;
    VI_Lighting_Base_Levels : ARRAY[1..16] OF BYTE;
    VI_Socket_States : ARRAY[1..36] OF BOOL;
    VI_Blinds_Positions : ARRAY[1..20] OF BYTE;
    VI_Active_Scenario : E_SCENARIO_TYPE;
  END_VAR
  VAR_OUTPUT
    VO_Modbus_Registers : ARRAY[0..200] OF WORD;  (* Расширенный диапазон *)
    VO_Lighting_Override : ARRAY[1..16] OF BYTE;
    VO_Socket_Override : ARRAY[1..36] OF BOOL;
    VO_Data_Ready : BOOL;
    VO_HMI_Status_Message : STRING(200);
  END_VAR
  VAR
    L_last_update_time : UDINT;
    L_i : INT;
    L_j : INT;
    L_idx : INT;
    L_tmp_word : WORD;
  END_VAR

            // Обновление данных Modbus (раз в 1 сек)
IF (VI_System_Time_MS - L_last_update_time) >= 1000 THEN
    L_last_update_time := VI_System_Time_MS;
    
    // 0: Статус ПЛК и Аварии
    L_tmp_word := 0;
    IF VI_Local_PLC_Role = E_PLC_ROLE.ROLE_ACTIVE THEN L_tmp_word := L_tmp_word OR 1; END_IF;
    IF VI_Security_Armed THEN L_tmp_word := L_tmp_word OR 2; END_IF;
    IF VI_Flood_Alarm_Active THEN L_tmp_word := L_tmp_word OR 4; END_IF;
    IF VI_Gas_Alarm_Active THEN L_tmp_word := L_tmp_word OR 8; END_IF;
    IF VI_Fire_Alarm_Active THEN L_tmp_word := L_tmp_word OR 16; END_IF;
    VO_Modbus_Registers[0] := L_tmp_word;

    // 1-16: Температуры пола (x10)
    FOR L_i := 1 TO 16 DO
        VO_Modbus_Registers[L_i] := TO_WORD(TO_INT(VI_FloorHeating_Temps[L_i] * 10.0));
    END_FOR;

    // 17-32: Температуры помещений (x10)
    FOR L_i := 1 TO 16 DO
        VO_Modbus_Registers[16 + L_i] := TO_WORD(TO_INT(VI_Room_Temps[L_i] * 10.0));
    END_FOR;

    // 33: Состояние клапанов зон (битовая маска 1-16)
    L_tmp_word := 0;
    FOR L_i := 1 TO 16 DO
        IF VI_Zone_Valve_States[L_i] THEN
            L_tmp_word := L_tmp_word OR SHL(TO_WORD(1), L_i - 1);
        END_IF;
    END_FOR;
    VO_Modbus_Registers[33] := L_tmp_word;

    // 34-38: Давление в коллекторах (x100)
    FOR L_i := 1 TO 5 DO
        VO_Modbus_Registers[33 + L_i] := TO_WORD(TO_INT(VI_Manifold_Pressures[L_i] * 100.0));
    END_FOR;

    // 40-55: Базовое освещение
    FOR L_i := 1 TO 16 DO
        VO_Modbus_Registers[39 + L_i] := TO_WORD(VI_Lighting_Base_Levels[L_i]);
    END_FOR;

    // 60-79: Положение штор (20 шт)
    FOR L_i := 1 TO 20 DO
        VO_Modbus_Registers[59 + L_i] := TO_WORD(VI_Blinds_Positions[L_i]);
    END_FOR;

    // 80-82: Розетки (битовая маска, 36 розеток -> 3 WORD)
    FOR L_i := 0 TO 2 DO
        L_tmp_word := 0;
        FOR L_j := 1 TO 16 DO
            L_idx := (L_i * 16) + L_j;
            IF L_idx <= 36 THEN
                IF VI_Socket_States[L_idx] THEN
                    L_tmp_word := L_tmp_word OR SHL(TO_WORD(1), L_j - 1);
                END_IF;
            END_IF;
        END_FOR;
        VO_Modbus_Registers[79 + L_i] := L_tmp_word;
    END_FOR;

    VO_Data_Ready := TRUE;
END_IF;

// Обработка входящих команд
IF VI_Command_Received AND (VI_Local_PLC_Role = E_PLC_ROLE.ROLE_ACTIVE) THEN
    CASE VI_Incoming_Command.command_type OF
        1: // Управление сценариями
            GVL_Vars.G_Current_Scenario := VI_Incoming_Command.target_scenario;
            VO_HMI_Status_Message := 'Gateway: Сценарий изменен';
        2: // Управление освещением
            IF (VI_Incoming_Command.target_zone >= 1) AND (VI_Incoming_Command.target_zone <= 16) THEN
                VO_Lighting_Override[VI_Incoming_Command.target_zone] := TO_BYTE(VI_Incoming_Command.target_value);
                VO_HMI_Status_Message := 'Gateway: Команда освещения принята';
            END_IF;
        3: // Розетки
            IF (VI_Incoming_Command.target_zone >= 1) AND (VI_Incoming_Command.target_zone <= 36) THEN
                VO_Socket_Override[VI_Incoming_Command.target_zone] := VI_Incoming_Command.target_on_off;
            END_IF;
        4: // Охрана
            // Логика постановки/снятия через PIN в FB_Security_System_Manager
            // Здесь можно только передать запрос
            VO_HMI_Status_Message := 'Gateway: Запрос охраны принят';
    END_CASE;
END_IF;

          
END_FUNCTION_BLOCK

FUNCTION_BLOCK FB_Heating_System_Manager
  VAR_INPUT
    VI_Maintenance_Zones : ARRAY[1..16] OF ST_Component_Maintenance;
    VI_Maintenance_Manifolds : ARRAY[1..5] OF ST_Component_Maintenance;
    VI_System_Time_MS : UDINT;
    VI_IsActivePLC : BOOL;
    VI_Outdoor_Temp : REAL;
    VI_Floor_Temps : ARRAY[1..16] OF REAL;
    VI_Room_Temps : ARRAY[1..16] OF REAL;
    VI_Config : ST_Heating_Config;
    VI_Manifold_Pressures : ARRAY[1..5] OF REAL;
    VI_Manifold_Currents : ARRAY[1..5] OF REAL;
    VI_Manifold_Temps_Supply : ARRAY[1..5] OF REAL;
    VI_Manifold_Temps_Return : ARRAY[1..5] OF REAL;
    VI_Boiler_Flame_Status : ARRAY[1..2] OF BOOL;
  END_VAR
  VAR_OUTPUT
    VO_Manifold_Valves : ARRAY[1..5] OF REAL;  (* 0-100% *)
    VO_Manifold_Pumps : ARRAY[1..5] OF BOOL;
    VO_Zone_Valves : ARRAY[1..16] OF BOOL;
    VO_Boiler_Enable : ARRAY[1..2] OF BOOL;
    VO_Boiler_Setpoint : ARRAY[1..2] OF REAL;  (* OpenTherm Setpoint *)
    VO_Status : ARRAY[1..5] OF ST_Manifold_Status;
    VO_Boiler_Status : ARRAY[1..2] OF ST_Boiler_Status;
  END_VAR
  VAR
    L_PID_Valves : ARRAY[1..5] OF FB_PID_Controller;
    L_Last_Boiler_Rotation : UDINT;
    L_Lead_Boiler : BYTE := 1;
    L_i : INT;
    L_Target_Supply_Temp : REAL;
    L_Demand_Power : REAL;
    L_Any_Zone_Active : ARRAY[1..5] OF BOOL;
    L_Overheat_Timer : ARRAY[1..16] OF TON;  (* ТЗ 2.5: Задержка перегрева *)
    L_Pump_Run_Timer : ARRAY[1..5] OF TON;  (* ТЗ 2.6: Диагностика *)
    L_Pump_Pause_Timer : ARRAY[1..5] OF TON;
    L_Pump_In_Pause : ARRAY[1..5] OF BOOL;
    L_Last_Scan_Time : UDINT;  (* ТЗ 2.8: Учет наработки *)
    L_Lifespan_S : REAL := 180000000;  (* 50,000 hours in seconds *)
  END_VAR

            // 1. Расчет целевой температуры подачи (ТЗ 2.3)
L_Target_Supply_Temp := 35.0;
IF VI_Config.Weather_Comp_Enabled AND VI_Outdoor_Temp < 15.0 THEN
    // Исправлено: убран множитель 10.0 согласно ТЗ 2.3
    L_Target_Supply_Temp := L_Target_Supply_Temp + (15.0 - VI_Outdoor_Temp) * VI_Config.Weather_Coef;
END_IF;
L_Target_Supply_Temp := LIMIT(20.0, L_Target_Supply_Temp, 45.0);

// 2. Управление зонами (ТЗ 1.1, 2.5)
FOR L_i := 1 TO 16 DO
    L_Overheat_Timer[L_i](IN := VI_Floor_Temps[L_i] > VI_Config.Overheat_Threshold, PT := T#60s);
    
    IF VI_Room_Temps[L_i] < (VI_Config.Target_Room_Temp - VI_Config.Hysteresis) THEN
        VO_Zone_Valves[L_i] := TRUE;
    ELSIF VI_Room_Temps[L_i] > (VI_Config.Target_Room_Temp + VI_Config.Hysteresis) THEN
        VO_Zone_Valves[L_i] := FALSE;
    END_IF;
    
    // Защита от перегрева с задержкой 60с (ТЗ 2.5)
    IF L_Overheat_Timer[L_i].Q THEN
        VO_Zone_Valves[L_i] := FALSE;
    END_IF;
END_FOR;

// 3. Активность коллекторов
L_Any_Zone_Active[1] := VO_Zone_Valves[1] OR VO_Zone_Valves[2];
L_Any_Zone_Active[2] := VO_Zone_Valves[3] OR VO_Zone_Valves[4] OR VO_Zone_Valves[5] OR VO_Zone_Valves[6];
L_Any_Zone_Active[3] := VO_Zone_Valves[7] OR VO_Zone_Valves[8] OR VO_Zone_Valves[9];
L_Any_Zone_Active[4] := VO_Zone_Valves[10] OR VO_Zone_Valves[11] OR VO_Zone_Valves[12];
L_Any_Zone_Active[5] := VO_Zone_Valves[13] OR VO_Zone_Valves[14] OR VO_Zone_Valves[15] OR VO_Zone_Valves[16];

// 4. Управление коллекторами (ТЗ 2.6, 12.2)
FOR L_i := 1 TO 5 DO
    L_PID_Valves[L_i](
        VI_SetPoint := L_Target_Supply_Temp,
        VI_ProcessValue := VI_Manifold_Temps_Supply[L_i],
        VI_Kp := 2.0, VI_Tn := 120.0, VI_Tv := 0.0,
        VI_Y_Min := 0.0, VI_Y_Max := 100.0, VI_Cycle_Time_S := 1.0,
        VO_Output => VO_Manifold_Valves[L_i]
    );

    // ТЗ 2.6: Пауза после 72 часов работы
    L_Pump_Run_Timer[L_i](IN := VO_Manifold_Pumps[L_i] AND NOT L_Pump_In_Pause[L_i], PT := T#72h);
    IF L_Pump_Run_Timer[L_i].Q THEN L_Pump_In_Pause[L_i] := TRUE; END_IF;
    
    L_Pump_Pause_Timer[L_i](IN := L_Pump_In_Pause[L_i], PT := T#1h);
    IF L_Pump_Pause_Timer[L_i].Q THEN L_Pump_In_Pause[L_i] := FALSE; END_IF;

    VO_Manifold_Pumps[L_i] := VI_IsActivePLC AND L_Any_Zone_Active[L_i] AND NOT L_Pump_In_Pause[L_i];

    // Защита от замерзания (ТЗ 2.4)
    IF VI_Outdoor_Temp < -5.0 OR VI_Manifold_Temps_Supply[L_i] < VI_Config.Freeze_Threshold THEN
        VO_Manifold_Pumps[L_i] := TRUE;
        VO_Manifold_Valves[L_i] := 100.0;
    END_IF;

    // Диагностика (ТЗ 2.6)
    VO_Status[L_i].Pump_On := VO_Manifold_Pumps[L_i];
    VO_Status[L_i].Pump_Current := VI_Manifold_Currents[L_i];
    VO_Status[L_i].Pressure := VI_Manifold_Pressures[L_i];
    VO_Status[L_i].Temp_Supply := VI_Manifold_Temps_Supply[L_i];
    VO_Status[L_i].Temp_Return := VI_Manifold_Temps_Return[L_i];
    VO_Status[L_i].Valve_Pos := VO_Manifold_Valves[L_i];
    
    // Контроль давления (1.5-2.5 бар) и Delta T (5-10C)
    IF VO_Manifold_Pumps[L_i] THEN
        IF VI_Manifold_Pressures[L_i] < 1.5 OR VI_Manifold_Pressures[L_i] > 2.5 THEN
            VO_Status[L_i].Error := TRUE; VO_Status[L_i].Error_ID := 16#E004; // Pressure Out of Range
        END_IF;
        // Исправлено: порог Delta T снижен до 10.0 согласно ТЗ 2.6
        IF (VI_Manifold_Temps_Supply[L_i] - VI_Manifold_Temps_Return[L_i]) > 10.0 THEN
            VO_Status[L_i].Error := TRUE; VO_Status[L_i].Error_ID := 16#E005; // High Delta T
        END_IF;
    END_IF;

    // Тестирование арматуры (ТЗ 12.2)
    IF (VI_System_Time_MS MOD 604800000) < 10000 THEN VO_Manifold_Valves[L_i] := 20.0; END_IF;
END_FOR;

// 5. Каскад котлов (ТЗ 2.8, 12.3)
L_Demand_Power := 0.0;
FOR L_i := 1 TO 5 DO IF VO_Manifold_Pumps[L_i] THEN L_Demand_Power := L_Demand_Power + VO_Manifold_Valves[L_i]; END_IF; END_FOR;
L_Demand_Power := L_Demand_Power / 5.0;

IF (VI_System_Time_MS - L_Last_Boiler_Rotation) > 604800000 THEN
    L_Last_Boiler_Rotation := VI_System_Time_MS;
    L_Lead_Boiler := SEL(L_Lead_Boiler = 1, 1, 2);
END_IF;

IF VI_IsActivePLC AND L_Demand_Power > 5.0 THEN
    VO_Boiler_Enable[L_Lead_Boiler] := TRUE;
    VO_Boiler_Setpoint[L_Lead_Boiler] := L_Target_Supply_Temp + 5.0; // OpenTherm Setpoint
    VO_Boiler_Enable[3 - L_Lead_Boiler] := (L_Demand_Power > 80.0);
    VO_Boiler_Setpoint[3 - L_Lead_Boiler] := SEL(L_Demand_Power > 80.0, 0.0, L_Target_Supply_Temp + 5.0);
ELSE
    VO_Boiler_Enable[1] := FALSE; VO_Boiler_Enable[2] := FALSE;
END_IF;

// Учет наработки (ТЗ 2.8, 12.3)
FOR L_i := 1 TO 2 DO
    IF VI_Boiler_Flame_Status[L_i] THEN
        VO_Boiler_Status[L_i].Work_Seconds := VO_Boiler_Status[L_i].Work_Seconds + 1; // Assuming 1s cycle for this FB or call
        VO_Boiler_Status[L_i].Work_Hours := TO_REAL(VO_Boiler_Status[L_i].Work_Seconds) / 3600.0;
        VO_Boiler_Status[L_i].Resource_Percent := (1.0 - (TO_REAL(VO_Boiler_Status[L_i].Work_Seconds) / L_Lifespan_S)) * 100.0;
    END_IF;
    VO_Boiler_Status[L_i].Running := VI_Boiler_Flame_Status[L_i];
END_FOR;

          
END_FUNCTION_BLOCK

FUNCTION_BLOCK FB_History_Manager
  VAR_INPUT
    VI_System_Time_MS : UDINT;
    VI_Write_Event : BOOL;
    VI_Event : ST_History_Record;
  END_VAR
  VAR_OUTPUT
    VO_Total_Events : UDINT;
  END_VAR
  VAR
    L_History_Buffer : ARRAY[1..100] OF ST_History_Record;
    L_Write_Idx : INT := 1;
  END_VAR

            IF VI_Write_Event THEN
    L_History_Buffer[L_Write_Idx] := VI_Event;
    L_History_Buffer[L_Write_Idx].timestamp_ms := VI_System_Time_MS;
    
    L_Write_Idx := (L_Write_Idx MOD 100) + 1;
    VO_Total_Events := VO_Total_Events + 1;
END_IF;

          
END_FUNCTION_BLOCK

FUNCTION_BLOCK FB_Lifetime_Predictor
  VAR_INPUT
    VI_Runtime_Hours : UDINT;
    VI_Start_Count : UDINT;
    VI_Nominal_Life : UDINT := 10000;
  END_VAR
  VAR_OUTPUT
    VO_Remaining_Percent : BYTE;
    VO_Maintenance_Req : BOOL;
  END_VAR

            // Упрощенная модель износа
IF VI_Nominal_Life > 0 THEN
    VO_Remaining_Percent := TO_BYTE(100 - (VI_Runtime_Hours * 100 / VI_Nominal_Life));
ELSE
    VO_Remaining_Percent := 0;
END_IF;

VO_Maintenance_Req := (VO_Remaining_Percent < 10);

          
END_FUNCTION_BLOCK

FUNCTION_BLOCK FB_Lighting_Blinds_Manager
  VAR_INPUT
    VI_System_Time_MS : UDINT;
    VI_IsActivePLC : BOOL;
    VI_Current_Scenario : E_SCENARIO_TYPE;
    VI_Away_Level : BYTE;  (* 1-Short, 2-Medium, 3-Long *)
    VI_Simulation_Active : BOOL;
    VI_Manual_Light_Override : ARRAY[1..16] OF BYTE;  (* 0-100 *)
    VI_Manual_Blinds_Override : ARRAY[1..20] OF BYTE;  (* 0-100 *)
    VI_Simulation_Lights : ARRAY[1..16] OF BOOL;
    VI_Physical_Switches : ARRAY[1..16] OF BOOL;  (* ТЗ 1.0 *)
    VI_Motion_Sensors : ARRAY[1..16] OF BOOL;  (* ТЗ 2.0 *)
    VI_Maintenance : ARRAY[1..16] OF ST_Component_Maintenance;  (* ТЗ 6.0 *)
  END_VAR
  VAR_OUTPUT
    VO_Lighting_Levels : ARRAY[1..16] OF BYTE;
    VO_Blinds_Positions : ARRAY[1..20] OF BYTE;
    VO_Wet_Zone_Light_Active : ARRAY[1..4] OF BOOL;  (* Для вентиляции (ТЗ 4.0) *)
  END_VAR
  VAR
    L_i : INT;
    L_Base_Light : BYTE;
    L_Base_Blinds : BYTE;
    L_Light_States : ARRAY[1..16] OF BOOL;
    L_Prev_Switches : ARRAY[1..16] OF BOOL;
    L_Motion_Timers : ARRAY[1..16] OF TON;
  END_VAR

            // 1. Определение базовых уровней по сценарию (ТЗ 7.1)
CASE VI_Current_Scenario OF
    E_SCENARIO_TYPE.SCENARIO_MORNING:
        L_Base_Light := 70;
        L_Base_Blinds := 80; // 80% открыты
    
    E_SCENARIO_TYPE.SCENARIO_EVENING:
        L_Base_Light := 40;
        L_Base_Blinds := 10; // 90% закрыты (10% открыты)
        
    E_SCENARIO_TYPE.SCENARIO_AWAY:
        L_Base_Light := 0;
        L_Base_Blinds := 0; // 100% закрыты
        
    ELSE
        L_Base_Light := 100;
        L_Base_Blinds := 100;
END_CASE;

// 2. Управление освещением
FOR L_i := 1 TO 16 DO
    // Приоритет 1: Физические выключатели (ТЗ 1.0)
    IF VI_Physical_Switches[L_i] AND NOT L_Prev_Switches[L_i] THEN
        L_Light_States[L_i] := NOT L_Light_States[L_i];
    END_IF;
    L_Prev_Switches[L_i] := VI_Physical_Switches[L_i];

    // Приоритет 2: Датчики движения (ТЗ 2.0)
    L_Motion_Timers[L_i](IN := VI_Motion_Sensors[L_i], PT := T#5m);
    IF VI_Motion_Sensors[L_i] THEN
        L_Light_States[L_i] := TRUE;
    ELSIF L_Motion_Timers[L_i].Q THEN
        L_Light_States[L_i] := FALSE;
    END_IF;

    // Приоритет 3: Симуляция (только в режиме Away)
    IF VI_Current_Scenario = E_SCENARIO_TYPE.SCENARIO_AWAY AND VI_Simulation_Active THEN
        L_Light_States[L_i] := VI_Simulation_Lights[L_i];
    END_IF;

    // Приоритет 4: Ремонт/Неисправность (ТЗ 6.0, 7.0)
    IF VI_Maintenance[L_i].Is_Faulty OR VI_Maintenance[L_i].Is_In_Maintenance THEN
        VO_Lighting_Levels[L_i] := REAL_TO_BYTE(VI_Maintenance[L_i].Fallback_Value);
    ELSE
        VO_Lighting_Levels[L_i] := SEL(L_Light_States[L_i], 0, L_Base_Light);
    END_IF;
    
    // 5. Мокрые зоны (допустим зоны 13-16 - санузлы)
    IF L_i >= 13 THEN
        VO_Wet_Zone_Light_Active[L_i - 12] := (VO_Lighting_Levels[L_i] > 10);
    END_IF;
END_FOR;

// 3. Управление шторами
FOR L_i := 1 TO 20 DO
    // Приоритет 1: Ручное управление
    IF VI_Manual_Blinds_Override[L_i] > 0 THEN
        VO_Blinds_Positions[L_i] := VI_Manual_Blinds_Override[L_i];
    // Приоритет 2: Сценарий
    ELSE
        VO_Blinds_Positions[L_i] := L_Base_Blinds;
    END_IF;
END_FOR;

          
END_FUNCTION_BLOCK

FUNCTION_BLOCK FB_Maintenance_Access
  VAR_INPUT
    VI_System_Time : UDINT;
    VI_Activate : BOOL;
    VI_Duration : UDINT := 60;  (* мин *)
  END_VAR
  VAR_OUTPUT
    VO_Active : BOOL;
    VO_Time_Left : UDINT;
  END_VAR
  VAR
    L_Start_Time : UDINT;
    L_elapsed : UDINT;
  END_VAR

            IF VI_Activate AND NOT VO_Active THEN
    VO_Active := TRUE;
    L_Start_Time := VI_System_Time;
END_IF;

IF VO_Active THEN
    L_elapsed := (VI_System_Time - L_Start_Time) / 60000;
    IF L_elapsed >= VI_Duration THEN
        VO_Active := FALSE;
    ELSE
        VO_Time_Left := VI_Duration - L_elapsed;
    END_IF;
END_IF;

          
END_FUNCTION_BLOCK

FUNCTION_BLOCK FB_Manifold_Mixing_Valve_Controller
  VAR_INPUT
    VI_Setpoint : REAL;
    VI_Actual : REAL;
  END_VAR
  VAR_OUTPUT
    VO_Valve_Pos : REAL;  (* 0-100% *)
  END_VAR

            // ПИД-регулятор (упрощенно для примера)
VO_Valve_Pos := (VI_Setpoint - VI_Actual) * 10.0;
IF VO_Valve_Pos > 100.0 THEN VO_Valve_Pos := 100.0;
ELSIF VO_Valve_Pos < 0.0 THEN VO_Valve_Pos := 0.0;
END_IF;

          
END_FUNCTION_BLOCK

FUNCTION_BLOCK FB_Manifold_Pump_Controller
  VAR_INPUT
    VI_Enable_Request : BOOL;
    VI_System_Time : UDINT;
    VI_Stop_Ramp_MS : UDINT := 5000;
  END_VAR
  VAR_OUTPUT
    VO_Speed_Percent : BYTE;
    VO_Running : BOOL;
  END_VAR
  VAR
    L_Stop_Start_Time : UDINT;
    L_Stopping : BOOL;
    L_elapsed : UDINT;
  END_VAR

            IF VI_Enable_Request THEN
    VO_Speed_Percent := 100;
    VO_Running := TRUE;
    L_Stopping := FALSE;
ELSE
    IF VO_Running AND NOT L_Stopping THEN
        L_Stopping := TRUE;
        L_Stop_Start_Time := VI_System_Time;
    END_IF;
    
    IF L_Stopping THEN
        L_elapsed := VI_System_Time - L_Stop_Start_Time;
        IF L_elapsed < VI_Stop_Ramp_MS THEN
            // Исправлено: защита от отрицательного значения
            VO_Speed_Percent := REAL_TO_BYTE(100.0 * (1.0 - TO_REAL(L_elapsed) / TO_REAL(VI_Stop_Ramp_MS)));
        ELSE
            VO_Speed_Percent := 0;
            VO_Running := FALSE;
            L_Stopping := FALSE;
        END_IF;
    END_IF;
END_IF;

          
END_FUNCTION_BLOCK

FUNCTION_BLOCK FB_Manual_Valve_Control
  VAR_INPUT
    VI_System_Time : UDINT;
    VI_Open_Req : BOOL;
    VI_Duration : UDINT := 5;  (* мин *)
  END_VAR
  VAR_OUTPUT
    VO_Open_Cmd : BOOL;
    VO_Time_Left : UDINT;
  END_VAR
  VAR
    L_Start_Time : UDINT;
    L_Active : BOOL;
    L_elapsed : UDINT;
  END_VAR

            // Логика ручного управления клапаном с таймером автозакрытия
IF VI_Open_Req AND NOT L_Active THEN
    L_Active := TRUE;
    L_Start_Time := VI_System_Time;
    VO_Open_Cmd := TRUE;
END_IF;

IF L_Active THEN
    // Расчет оставшегося времени в минутах
    L_elapsed := (VI_System_Time - L_Start_Time) / 60000;
    IF L_elapsed >= VI_Duration THEN
        L_Active := FALSE;
        VO_Open_Cmd := FALSE;
    ELSE
        VO_Time_Left := VI_Duration - L_elapsed;
    END_IF;
ELSE
    VO_Time_Left := 0;
END_IF;

          
END_FUNCTION_BLOCK

FUNCTION_BLOCK FB_NVRAM_Manager
  VAR_INPUT
    VI_Command : BYTE;  (* 1=WRITE, 2=READ, 3=FORMAT *)
    VI_RecordIndex : INT;
    VI_DataPtr : POINTER TO BYTE;
    VI_DataSize : UDINT;  (* КРИТИЧНО: используем этот размер вместо SIZEOF *)
    VI_System_Time_MS : UDINT;
    VI_Operator_ID : STRING(10);
    VI_IsActivePLC : BOOL;
    VI_TwoPersonConfirmation : BOOL;
  END_VAR
  VAR_OUTPUT
    VO_Done : BOOL;
    VO_Error : UDINT;
    VO_ErrorID : UDINT;
    VO_ReadDataPtr : POINTER TO BYTE;
    VO_HMI_Status_Message : STRING(200);
  END_VAR
  VAR
    L_state : BYTE;
    L_step : UDINT;
    L_temp_buffer : ARRAY[1..132] OF BYTE;
    L_crc32 : FB_CRC32_Calculator;
    L_confirm_start_time : UDINT;
    L_cmd_copy : BYTE;
    L_prev_Command : BYTE;
    L_i : UDINT;
    L_current_time : UDINT;
    L_cmd_rising : BOOL;
    L_data_crc : DWORD;
    L_FileHandle : RTS_IEC_HANDLE;
    L_FileName : STRING := '/home/root/nvram_data.bin';
    L_FileResult : RTS_IEC_RESULT;
    L_BytesProcessed : UDINT;
    L_BackupIdx : INT := 1;  (* Для ротации *)
    L_Offset : DINT;
  END_VAR
  VAR CONSTANT
    C_MAGIC_NUMBER : UDINT := 16#534D5254;  (* "SMRT" *)
    C_STRUCT_VERSION : UINT := 21;  (* ТЗ v21.0 *)
    C_NVRAM_BASE_ADDR : UDINT := 16#20000;
    C_HEADER_SIZE : UDINT := 12;
    C_RECORD_SIZE : UDINT := 128;
    C_RECORD_TOTAL_SIZE : UDINT := 132;
    C_MAX_RECORDS : UDINT := 96;
    C_TWO_PERSON_TIMEOUT_MS : UDINT := 120000;
  END_VAR

            // Логика выполнения
L_current_time := VI_System_Time_MS;

// Детекция фронта команды
L_cmd_rising := (VI_Command <> 0) AND (L_prev_Command = 0);
L_prev_Command := VI_Command;

CASE L_state OF
    0: // ОЖИДАНИЕ (IDLE)
        IF L_cmd_rising THEN
            VO_Done := FALSE;
            VO_Error := 0;
            
            // Валидация индекса
            IF (VI_RecordIndex < 1) OR (TO_UDINT(VI_RecordIndex) > C_MAX_RECORDS) THEN
                VO_Error := 16#1501;
                VO_HMI_Status_Message := 'NVRAM: Неверный индекс записи';
                VO_Done := TRUE;
                RETURN;
            END_IF;

            // Валидация указателя
            IF VI_DataPtr = 0 THEN
                VO_Error := 16#150A;
                VO_HMI_Status_Message := 'NVRAM: Нулевой указатель данных';
                VO_Done := TRUE;
                RETURN;
            END_IF;

            IF VI_Command = 1 THEN // ЗАПИСЬ (WRITE)
                IF NOT VI_IsActivePLC THEN
                    VO_Error := 16#1509;
                    VO_HMI_Status_Message := 'NVRAM: Запись запрещена (STANDBY)';
                    VO_Done := TRUE;
                ELSIF VI_DataSize > C_RECORD_SIZE THEN
                    VO_Error := 16#150B;
                    VO_HMI_Status_Message := 'NVRAM: Размер данных больше 128 байт';
                    VO_Done := TRUE;
                ELSE
                    L_state := 1; // Переход к записи
                    L_step := 0;
                END_IF;
            ELSIF VI_Command = 2 THEN // ЧТЕНИЕ (READ)
                L_state := 2; // Переход к чтению
                L_step := 0;
            END_IF;
        END_IF;

    1: // ЗАПИСЬ_ЗАПИСИ (WRITE_RECORD)
        CASE L_step OF
            0: // Подготовка буфера и расчет CRC
                FOR L_i := 0 TO C_RECORD_SIZE - 1 DO
                    IF L_i < VI_DataSize THEN
                        L_temp_buffer[TO_INT(L_i + 1)] := VI_DataPtr[TO_INT(L_i)];
                    ELSE
                        L_temp_buffer[TO_INT(L_i + 1)] := 16#00;
                    END_IF;
                END_FOR;
                L_data_crc := L_crc32.Calculate(ADR(L_temp_buffer[1]), C_RECORD_SIZE);
                L_step := 1;
                
            1: // Открытие файла для записи
                L_FileHandle := SysFileOpen(L_FileName, AM_WRITE, ADR(L_FileResult));
                IF L_FileResult = 0 THEN
                    L_step := 2;
                ELSE
                    VO_Error := 16#150C;
                    L_state := 0;
                END_IF;
                
            2: // Позиционирование и запись
                L_Offset := TO_DINT(VI_RecordIndex - 1) * TO_DINT(C_RECORD_TOTAL_SIZE);
                L_FileResult := SysFileSetPos(L_FileHandle, TO_UDINT(L_Offset));
                L_BytesProcessed := TO_UDINT(SysFileWrite(L_FileHandle, ADR(L_temp_buffer[1]), TO_UDINT(C_RECORD_TOTAL_SIZE), ADR(L_FileResult)));
                L_FileResult := SysFileClose(L_FileHandle);
                VO_Done := TRUE;
                L_state := 0;
        END_CASE;

    2: // ЧТЕНИЕ_ЗАПИСИ (READ_RECORD)
        CASE L_step OF
            0: // Открытие файла для чтения
                L_FileHandle := SysFileOpen(L_FileName, AM_READ, ADR(L_FileResult));
                IF L_FileResult = 0 THEN
                    L_step := 1;
                ELSE
                    VO_Error := 16#150D;
                    L_state := 0;
                END_IF;
                
            1: // Чтение данных
                L_Offset := TO_DINT(VI_RecordIndex - 1) * TO_DINT(C_RECORD_TOTAL_SIZE);
                L_FileResult := SysFileSetPos(L_FileHandle, TO_UDINT(L_Offset));
                L_BytesProcessed := TO_UDINT(SysFileRead(L_FileHandle, ADR(L_temp_buffer[1]), TO_UDINT(C_RECORD_TOTAL_SIZE), ADR(L_FileResult)));
                L_FileResult := SysFileClose(L_FileHandle);
                
                // Копирование в выходной указатель
                FOR L_i := 0 TO C_RECORD_SIZE - 1 DO
                    IF L_i < VI_DataSize THEN
                        VI_DataPtr[TO_INT(L_i)] := L_temp_buffer[TO_INT(L_i + 1)];
                    END_IF;
                END_FOR;
                VO_ReadDataPtr := VI_DataPtr;
                VO_Done := TRUE;
                L_state := 0;
        END_CASE;
END_CASE;

          
END_FUNCTION_BLOCK

FUNCTION_BLOCK FB_Outdoor_Lighting_Controller
  VAR_INPUT
    VI_Ambient_Lux : REAL;
    VI_Motion : BOOL;
    VI_Security : BOOL;
  END_VAR
  VAR_OUTPUT
    VO_Light_On : BOOL;
  END_VAR

            IF VI_Security AND VI_Motion THEN
    VO_Light_On := TRUE; // Тревожное освещение
ELSIF VI_Ambient_Lux < 50.0 THEN
    VO_Light_On := TRUE; // Ночное освещение
ELSE
    VO_Light_On := FALSE;
END_IF;

          
END_FUNCTION_BLOCK

FUNCTION_BLOCK FB_PID_Controller
  VAR_INPUT
    VI_SetPoint : REAL;  (* Уставка *)
    VI_ProcessValue : REAL;  (* Текущее значение *)
    VI_Kp : REAL;  (* Коэффициент усиления *)
    VI_Tn : REAL;  (* Время интегрирования (сек) *)
    VI_Tv : REAL;  (* Время дифференцирования (сек) *)
    VI_Y_Min : REAL := 0;  (* Минимальный выход *)
    VI_Y_Max : REAL := 100;  (* Максимальный выход *)
    VI_Manual_Mode : BOOL;  (* Ручной режим *)
    VI_Manual_Value : REAL;  (* Значение в ручном режиме *)
    VI_Deadband : REAL := 0.1;  (* Мертвая зона *)
    VI_Cycle_Time_S : REAL := 0.01;  (* Время цикла задачи в секундах *)
    VI_Reset : BOOL;  (* Сброс интегральной составляющей *)
  END_VAR
  VAR_OUTPUT
    VO_Output : REAL;  (* Выход регулятора *)
    VO_Error : REAL;  (* Ошибка рассогласования *)
    VO_Limiting : BOOL;  (* Флаг ограничения выхода (Anti-windup) *)
  END_VAR
  VAR
    L_Integral_Sum : REAL;  (* Интегральная сумма *)
    L_Prev_Error : REAL;  (* Предыдущая ошибка *)
    L_Derivative : REAL;  (* Дифференциальная составляющая *)
    L_Output_Raw : REAL;  (* Сырой выход до ограничения *)
  END_VAR

            // Расчет ошибки
VO_Error := VI_SetPoint - VI_ProcessValue;

// Проверка мертвой зоны
IF ABS(VO_Error) < VI_Deadband THEN
    VO_Error := 0.0;
END_IF;

IF VI_Reset THEN
    L_Integral_Sum := 0.0;
    L_Prev_Error := 0.0;
    VO_Output := 0.0;
    RETURN;
END_IF;

IF VI_Manual_Mode THEN
    VO_Output := VI_Manual_Value;
    L_Integral_Sum := VO_Output; // Безударный переход
    RETURN;
END_IF;

// Пропорциональная составляющая
L_Output_Raw := VI_Kp * VO_Error;

// Интегральная составляющая (Метод трапеций)
IF VI_Tn > 0.0 THEN
    // Anti-windup: не накапливаем интеграл, если выход уже на пределе и ошибка того же знака
    IF NOT VO_Limiting OR (VO_Error > 0.0 AND L_Output_Raw < VI_Y_Max) OR (VO_Error < 0.0 AND L_Output_Raw > VI_Y_Min) THEN
        L_Integral_Sum := L_Integral_Sum + (VI_Kp / VI_Tn) * VO_Error * VI_Cycle_Time_S;
    END_IF;
    L_Output_Raw := L_Output_Raw + L_Integral_Sum;
END_IF;

// Дифференциальная составляющая
IF VI_Tv > 0.0 THEN
    L_Derivative := (VO_Error - L_Prev_Error) / VI_Cycle_Time_S;
    L_Output_Raw := L_Output_Raw + VI_Kp * VI_Tv * L_Derivative;
END_IF;

L_Prev_Error := VO_Error;

// Ограничение выхода
IF L_Output_Raw > VI_Y_Max THEN
    VO_Output := VI_Y_Max;
    VO_Limiting := TRUE;
ELSIF L_Output_Raw < VI_Y_Min THEN
    VO_Output := VI_Y_Min;
    VO_Limiting := TRUE;
ELSE
    VO_Output := L_Output_Raw;
    VO_Limiting := FALSE;
END_IF;

          
END_FUNCTION_BLOCK

FUNCTION_BLOCK FB_PLC_Heartbeat
  VAR_INPUT
    VI_Local_ID : BYTE;
    VI_System_Time : UDINT;
    VI_Remote_Pulse : BOOL;
    VI_Remote_Is_Active : BOOL;  (* ТЗ 8.3: Уровень 2 - проверка роли партнера *)
    VI_Gateway_Ping_OK : BOOL;  (* ТЗ 8.3: Уровень 3 - пинг шлюза *)
  END_VAR
  VAR_OUTPUT
    VO_Is_Active : BOOL;
    VO_RTT_MS : UDINT;
    VO_Loss_Count : UDINT;  (* ТЗ 8.4: Статистика потерь *)
    VO_Max_RTT : UDINT;  (* ТЗ 8.4: Макс. задержка *)
  END_VAR
  VAR
    L_Last_Pulse : BOOL;
    L_Last_Pulse_Time : UDINT;
    L_Timeout : UDINT := 500;  (* ТЗ 8.1: 500 мс *)
    L_Pulse_Send_Time : UDINT;
    L_Loss_Timer : TON;
  END_VAR

            // 1. Мониторинг пульса и RTT (ТЗ 8.4)
IF VI_Remote_Pulse <> L_Last_Pulse THEN
    VO_RTT_MS := VI_System_Time - L_Last_Pulse_Time;
    IF VO_RTT_MS > VO_Max_RTT THEN VO_Max_RTT := VO_RTT_MS; END_IF;
    L_Last_Pulse := VI_Remote_Pulse;
    L_Last_Pulse_Time := VI_System_Time;
END_IF;

L_Loss_Timer(IN := (VI_System_Time - L_Last_Pulse_Time) > L_Timeout, PT := T#1s);
IF L_Loss_Timer.Q THEN 
    VO_Loss_Count := VO_Loss_Count + 1; 
    L_Loss_Timer(IN := FALSE); 
END_IF;

// 2. Логика активности и защита от раскола мозга (ТЗ 8.3)
// Уровень 1: Тайм-аут пульса
IF (VI_System_Time - L_Last_Pulse_Time) < L_Timeout THEN
    // Уровень 2: Если партнер заявляет, что он активен, и у него приоритет (ID=1)
    IF VI_Remote_Is_Active AND VI_Local_ID = 2 THEN
        VO_Is_Active := FALSE;
    ELSE
        // Приоритет у ПЛК A (ID=1)
        VO_Is_Active := (VI_Local_ID = 1);
    END_IF;
ELSE
    // Уровень 3: Если связи нет, проверяем доступность шлюза
    VO_Is_Active := VI_Gateway_Ping_OK OR (VI_Local_ID = 1);
END_IF;

          
END_FUNCTION_BLOCK

FUNCTION_BLOCK FB_Pre_Departure_Heating
  VAR_INPUT
    VI_Departure_Time : UDINT;
    VI_System_Time : UDINT;
    VI_Selected : ARRAY[1..16] OF BOOL;
  END_VAR
  VAR_OUTPUT
    VO_Heating_Active : BOOL;
    VO_Setpoints : ARRAY[1..16] OF REAL;
  END_VAR
  VAR
    L_i : INT;
  END_VAR

            // Запуск за 3 часа (10800000 мс)
IF (VI_Departure_Time - VI_System_Time) < 10800000 THEN
    VO_Heating_Active := TRUE;
    FOR L_i := 1 TO 16 DO
        IF VI_Selected[L_i] THEN VO_Setpoints[L_i] := 22.0; END_IF;
    END_FOR;
ELSE
    VO_Heating_Active := FALSE;
END_IF;

          
END_FUNCTION_BLOCK

FUNCTION_BLOCK FB_Presence_Playback
  VAR_INPUT
    VI_Mode_Record : BOOL;  (* TRUE - записываем, FALSE - воспроизводим *)
    VI_Light_Inputs : ARRAY[1..16] OF BOOL;
    VI_Time_Index : UDINT;  (* Индекс времени в рамках недели (мс) *)
  END_VAR
  VAR_OUTPUT
    VO_Light_Outputs : ARRAY[1..16] OF BOOL;
  END_VAR
  VAR
    L_History : ARRAY[0..1007] OF WORD;  (* 168 часов * 6 записей в час = 1008 записей (битовая маска 16 ламп) *)
    L_Current_Slot : UDINT;
    L_i : INT;
  END_VAR

            L_Current_Slot := (VI_Time_Index / 600000) MOD 1008; // Слот каждые 10 минут

IF VI_Mode_Record THEN
    // Запись текущего состояния в слот
    L_History[L_Current_Slot] := 0;
    FOR L_i := 1 TO 16 DO
        IF VI_Light_Inputs[L_i] THEN
            L_History[L_Current_Slot] := L_History[L_Current_Slot] OR SHL(WORD#1, L_i-1);
        END_IF;
    END_FOR;
ELSE
    // Воспроизведение из слота
    FOR L_i := 1 TO 16 DO
        VO_Light_Outputs[L_i] := (L_History[L_Current_Slot] AND SHL(WORD#1, L_i-1)) <> 0;
    END_FOR;
END_IF;

          
END_FUNCTION_BLOCK

FUNCTION_BLOCK FB_Presence_Simulator
  VAR_INPUT
    VI_Enabled : BOOL;
    VI_Intensity : REAL;
    VI_System_Time : UDINT;
    VI_Use_Playback : BOOL;  (* Новый режим воспроизведения *)
  END_VAR
  VAR_OUTPUT
    VO_Light_States : ARRAY[1..16] OF BOOL;
  END_VAR
  VAR
    fbPlayback : FB_Presence_Playback;
  END_VAR

            IF VI_Enabled THEN
    IF VI_Use_Playback THEN
        fbPlayback(VI_Mode_Record := FALSE, VI_Time_Index := VI_System_Time MOD 604800000, VO_Light_Outputs => VO_Light_States);
    ELSE
        // Старая логика случайной симуляции
        VO_Light_States[1] := (VI_System_Time MOD 100000 > 50000);
    END_IF;
END_IF;

          
END_FUNCTION_BLOCK

FUNCTION_BLOCK FB_Random_Generator
  VAR
    L_seed : UDINT := 1;
  END_VAR
  VAR CONSTANT
    C_LCG_MULTIPLIER : UDINT := 1664525;
    C_LCG_INCREMENT : UDINT := 1013904223;
    C_LCG_MODULUS : LREAL := 4294967296;
  END_VAR

            
          

METHOD Random_Int_Range : UDINT
  VAR_INPUT
    VI_min : UDINT;
    VI_max : UDINT;
  END_VAR
  VAR
    L_range : UDINT;
    L_rand_factor : LREAL;
  END_VAR
                  L_seed := (C_LCG_MULTIPLIER * L_seed) + C_LCG_INCREMENT;

IF VI_max > VI_min THEN
        L_range := VI_max - VI_min;
        // Используем LREAL для точности и исключения выхода за границу
        L_rand_factor := TO_LREAL(L_seed) / C_LCG_MODULUS;
        Random_Int_Range := VI_min + TO_UDINT(L_rand_factor * TO_LREAL(L_range + 1));
        
        // Финальная защита от переполнения
        IF Random_Int_Range > VI_max THEN
            Random_Int_Range := VI_max;
        END_IF;
    ELSE
        Random_Int_Range := VI_min;
    END_IF;
                
END_METHOD
END_FUNCTION_BLOCK

FUNCTION_BLOCK FB_Scenario_Manager
  VAR_INPUT
    VI_System_Time_MS : UDINT;
    VI_Activate_Request : E_SCENARIO_TYPE;
    VI_IsActivePLC : BOOL;
  END_VAR
  VAR_OUTPUT
    VO_Current_Scenario : E_SCENARIO_TYPE;
    VO_Status_Msg : STRING(200);
  END_VAR

            IF VI_IsActivePLC AND (VI_Activate_Request <> VO_Current_Scenario) THEN
    // Логика переключения сценариев
    VO_Current_Scenario := VI_Activate_Request;
    
    CASE VO_Current_Scenario OF
        E_SCENARIO_TYPE.SCENARIO_NONE:
            VO_Status_Msg := 'Сценарии отключены';
        E_SCENARIO_TYPE.SCENARIO_AWAY:
            VO_Status_Msg := 'Активирован сценарий: Вне дома (Охрана + Энергосбережение)';
        E_SCENARIO_TYPE.SCENARIO_SLEEP:
            VO_Status_Msg := 'Активирован сценарий: Сон (Ночное освещение + Климат)';
        E_SCENARIO_TYPE.SCENARIO_PRESENCE:
            VO_Status_Msg := 'Активирован сценарий: Имитация присутствия';
    END_CASE;
END_IF;

          
END_FUNCTION_BLOCK

FUNCTION_BLOCK FB_Scenario_Transition_Controller
  VAR_INPUT
    VI_System_Time : UDINT;
    VI_Start_Time : UDINT;
    VI_Min_Dur : UDINT := 300000;  (* 5 мин *)
  END_VAR
  VAR_OUTPUT
    VO_Allowed : BOOL;
  END_VAR

            VO_Allowed := (VI_System_Time - VI_Start_Time) >= VI_Min_Dur;

          
END_FUNCTION_BLOCK

FUNCTION_BLOCK FB_Security_Alarm
  VAR_INPUT
    VI_IsActivePLC : BOOL;
    VI_Assigned_DoorWindow_Open : ARRAY[1..20] OF BOOL;
    VI_Assigned_GlassBreak : ARRAY[1..12] OF BOOL;
  END_VAR
  VAR_OUTPUT
    VO_Alarm_Active : BOOL;
    VO_Status_Msg : STRING(200);
  END_VAR

            VO_Alarm_Active := CheckPerimeter();

IF VO_Alarm_Active THEN
    VO_Status_Msg := 'ТРЕВОГА: НАРУШЕН ПЕРИМЕТР';
ELSE
    VO_Status_Msg := 'Периметр в норме';
END_IF;


          

METHOD CheckPerimeter : BOOL
  VAR
    L_i : INT;
  END_VAR
                  CheckPerimeter := FALSE;
// Проверка окон
FOR L_i := 1 TO 20 DO
    IF VI_Assigned_DoorWindow_Open[L_i] THEN
        CheckPerimeter := TRUE;
        RETURN;
    END_IF;
END_FOR;
// Проверка стекол
FOR L_i := 1 TO 12 DO
    IF VI_Assigned_GlassBreak[L_i] THEN
        CheckPerimeter := TRUE;
        RETURN;
    END_IF;
END_FOR;
                
END_METHOD
END_FUNCTION_BLOCK

FUNCTION_BLOCK FB_Security_System
  VAR_INPUT
    VI_System_Time : UDINT;
    VI_Sensors_Open : ARRAY[1..15] OF BOOL;
    VI_Sensors_Glass : ARRAY[1..15] OF BOOL;
    VI_Grouped_2F : BOOL;
    VI_PIN_Code : STRING(4);
    VI_Arm_Request : BOOL;
  END_VAR
  VAR_OUTPUT
    VO_Alarm_Active : BOOL;
    VO_Alarm_Level : E_ALERT_PRIORITY;
    VO_Status : BYTE;  (* 0-Disarmed, 1-Arming, 2-Armed, 3-Alarm *)
  END_VAR
  VAR
    L_Last_Trigger_Time : UDINT;
    L_Trigger_Count : INT;
    L_i : INT;
  END_VAR

            L_Trigger_Count := 0;
FOR L_i := 1 TO 15 DO
    IF VI_Sensors_Open[L_i] OR VI_Sensors_Glass[L_i] THEN
        L_Trigger_Count := L_Trigger_Count + 1;
    END_IF;
END_FOR;
IF VI_Grouped_2F THEN L_Trigger_Count := L_Trigger_Count + 1; END_IF;

// Логика п. 3.3: Комбинированные события (>=2 датчиков за 10 сек)
IF L_Trigger_Count >= 2 THEN
    IF (VI_System_Time - L_Last_Trigger_Time) < 10000 THEN
        VO_Alarm_Level := E_ALERT_PRIORITY.ALERT_PRIORITY_CRITICAL;
        VO_Alarm_Active := TRUE;
    END_IF;
    L_Last_Trigger_Time := VI_System_Time;
END_IF;

          
END_FUNCTION_BLOCK

FUNCTION_BLOCK FB_Security_System_Manager
  VAR_INPUT
    VI_System_Time_MS : UDINT;
    VI_IsActivePLC : BOOL;
    VI_Opening_Sensors : ARRAY[1..15] OF BOOL;
    VI_GlassBreak_Sensors : ARRAY[1..15] OF BOOL;
    VI_PIN_Input : STRING(4);
    VI_PIN_Submit : BOOL;
    VI_Config : ST_Security_Config;
    VI_Outdoor_Lux : REAL;
    VI_Motion_Corridor : BOOL;
    VI_Acknowledge_Open_Windows : BOOL;  (* ТЗ 3.8 *)
    VI_Group_2F_Open : BOOL;  (* ТЗ 3.1 (7 окон -> 1 канал) *)
    VI_Group_2F_Glass : BOOL;  (* ТЗ 3.2 *)
  END_VAR
  VAR_OUTPUT
    VO_Armed : BOOL;
    VO_Alarm_Active : BOOL;
    VO_Entry_Delay_Active : BOOL;
    VO_Time_To_Alarm_S : UINT;
    VO_Away_Level : BYTE;  (* 1-Short, 2-Medium, 3-Long *)
    VO_Light_Corridor : BOOL;
    VO_Light_Stairs_Dim : BYTE;
    VO_Status_Msg : STRING(200);
    VO_Long_Away_Req : BOOL;  (* ТЗ 3.6: При тревоге -> долгосрочный отъезд *)
  END_VAR
  VAR
    L_State : BYTE;  (* 0-Disarmed, 1-Armed, 2-EntryDelay, 3-Alarm, 4-ConfirmWait *)
    L_Attempts : UINT;
    L_Entry_Start_Time : UDINT;
    L_Away_Start_Time : UDINT;
    L_Confirm_Start_Time : UDINT;
    L_Last_Trigger_Time : UDINT;
    L_i : INT;
    L_Any_Sensor_Open : BOOL;
    L_Any_Glass_Broken : BOOL;
    L_Trigger_Count : UINT;  (* ТЗ 3.3: Комбинированные события (>=2 за 10с) *)
    L_Trigger_Timer : TON;
    L_Last_Sensors : ARRAY[1..32] OF BOOL;
    L_Glass_Threshold_Multiplier : REAL := 1;  (* ТЗ 3.8: Снижение порога *)
  END_VAR

            // 1. Мониторинг датчиков
L_Any_Sensor_Open := VI_Group_2F_Open;
FOR L_i := 1 TO 15 DO IF VI_Opening_Sensors[L_i] THEN L_Any_Sensor_Open := TRUE; EXIT; END_IF; END_FOR;

L_Any_Glass_Broken := VI_Group_2F_Glass;
FOR L_i := 1 TO 15 DO IF VI_GlassBreak_Sensors[L_i] THEN L_Any_Glass_Broken := TRUE; EXIT; END_IF; END_FOR;

// ТЗ 3.3: Подсчет срабатываний за 10с
L_Trigger_Timer(IN := L_Trigger_Count > 0, PT := T#10s);
IF L_Trigger_Timer.Q THEN L_Trigger_Count := 0; END_IF;

FOR L_i := 1 TO 15 DO
    IF VI_Opening_Sensors[L_i] AND NOT L_Last_Sensors[L_i] THEN L_Trigger_Count := L_Trigger_Count + 1; END_IF;
    L_Last_Sensors[L_i] := VI_Opening_Sensors[L_i];
    
    IF VI_GlassBreak_Sensors[L_i] AND NOT L_Last_Sensors[15 + L_i] THEN L_Trigger_Count := L_Trigger_Count + 1; END_IF;
    L_Last_Sensors[15 + L_i] := VI_GlassBreak_Sensors[L_i];
END_FOR;
// Групповые датчики тоже участвуют в подсчете
IF VI_Group_2F_Open AND NOT L_Last_Sensors[31] THEN L_Trigger_Count := L_Trigger_Count + 1; END_IF;
L_Last_Sensors[31] := VI_Group_2F_Open;
IF VI_Group_2F_Glass AND NOT L_Last_Sensors[32] THEN L_Trigger_Count := L_Trigger_Count + 1; END_IF;
L_Last_Sensors[32] := VI_Group_2F_Glass;

// ТЗ 3.8: Снижение порога на 20% (увеличиваем чувствительность)
L_Glass_Threshold_Multiplier := SEL(VI_Acknowledge_Open_Windows, 1.0, 0.8);

// 2. Логика состояний
CASE L_State OF
    0: // Снято с охраны
        VO_Armed := FALSE; VO_Alarm_Active := FALSE; VO_Entry_Delay_Active := FALSE; VO_Long_Away_Req := FALSE;
        IF VI_PIN_Submit AND VI_PIN_Input = VI_Config.PIN_Code THEN
            IF NOT L_Any_Sensor_Open OR VI_Acknowledge_Open_Windows THEN
                IF VI_Config.Two_Stage_Mode THEN
                    L_State := 4; L_Confirm_Start_Time := VI_System_Time_MS;
                    VO_Status_Msg := 'Ожидание второго этапа подтверждения';
                ELSE
                    L_State := 1; L_Away_Start_Time := VI_System_Time_MS; L_Attempts := 0;
                    VO_Status_Msg := 'Система поставлена на охрану';
                END_IF;
            ELSE
                VO_Status_Msg := 'Ошибка: Обнаружены открытые окна/двери';
            END_IF;
        END_IF;

    4: // Ожидание второго этапа (ТЗ 3.4)
        IF (VI_System_Time_MS - L_Confirm_Start_Time) / 1000 >= VI_Config.Confirmation_Timeout_S THEN
            L_State := 0; VO_Status_Msg := 'Таймаут подтверждения постановки';
        ELSIF VI_PIN_Submit AND VI_PIN_Input = VI_Config.PIN_Code THEN
             L_State := 1; L_Away_Start_Time := VI_System_Time_MS; L_Attempts := 0;
             VO_Status_Msg := 'Система поставлена на охрану (2 этапа)';
        END_IF;

    1: // На охране
        VO_Armed := TRUE;
        // ТЗ 3.3: Немедленная тревога если >=2 датчика за 10с
        IF L_Trigger_Count >= 2 THEN
            L_State := 3;
        ELSIF L_Any_Sensor_Open OR L_Any_Glass_Broken THEN
            L_State := 2; L_Entry_Start_Time := VI_System_Time_MS;
        END_IF;

    2: // Задержка входа (ТЗ 3.3)
        VO_Entry_Delay_Active := TRUE;
        VO_Time_To_Alarm_S := TO_UINT(VI_Config.Entry_Delay_S - (VI_System_Time_MS - L_Entry_Start_Time) / 1000);
        IF VI_PIN_Submit THEN
            IF VI_PIN_Input = VI_Config.PIN_Code THEN L_State := 0; VO_Status_Msg := 'Система снята с охраны';
            ELSE
                L_Attempts := L_Attempts + 1;
                IF L_Attempts >= VI_Config.Max_Attempts THEN L_State := 3; END_IF;
            END_IF;
        END_IF;
        IF (VI_System_Time_MS - L_Entry_Start_Time) / 1000 >= VI_Config.Entry_Delay_S THEN L_State := 3; END_IF;

    3: // Тревога
        VO_Alarm_Active := TRUE;
        VO_Long_Away_Req := TRUE; // ТЗ 3.6: При тревоге -> долгосрочный отъезд
        VO_Status_Msg := 'ТРЕВОГА: НАРУШЕНИЕ ПЕРИМЕТРА';
        IF VI_PIN_Submit AND VI_PIN_Input = VI_Config.PIN_Code THEN L_State := 0; VO_Status_Msg := 'Тревога сброшена'; END_IF;
END_CASE;

// 3. Уровни отъезда (ТЗ 3.5)
IF L_State <> 0 THEN
    L_Last_Trigger_Time := (VI_System_Time_MS - L_Away_Start_Time) / 3600000; // Часы
    IF L_Last_Trigger_Time < 2 THEN VO_Away_Level := 1;
    ELSIF L_Last_Trigger_Time < 72 THEN VO_Away_Level := 2;
    ELSE VO_Away_Level := 3; END_IF;
ELSE VO_Away_Level := 0; END_IF;

// 4. Интеграция с освещением (ТЗ 3.9)
IF (VI_Outdoor_Lux < 50.0 OR (TOD_TO_UDINT(UDINT_TO_TOD(VI_System_Time_MS)) > 64800000 OR TOD_TO_UDINT(UDINT_TO_TOD(VI_System_Time_MS)) < 28800000)) THEN
    IF VI_Motion_Corridor OR (L_State = 2) THEN VO_Light_Corridor := TRUE; VO_Light_Stairs_Dim := 30;
    ELSE VO_Light_Corridor := FALSE; VO_Light_Stairs_Dim := 0; END_IF;
END_IF;

          
END_FUNCTION_BLOCK

FUNCTION_BLOCK FB_Sensor_Calibration_Processor
  VAR_INPUT
    VI_Raw_Value : REAL;
    VI_Calib_Record : ST_Sensor_Calibration_Record;
  END_VAR
  VAR_OUTPUT
    VO_Calibrated_Value : REAL;
  END_VAR

            // Формула: (Сырое значение * Множитель) + Смещение
VO_Calibrated_Value := (VI_Raw_Value * VI_Calib_Record.multiplier) + VI_Calib_Record.offset;

          
END_FUNCTION_BLOCK

FUNCTION_BLOCK FB_Sensor_Distribution
  VAR_INPUT
    VI_Local_PLC_ID : BYTE;  (* 1=A, 2=B *)
    VI_Raw_Sensors : ARRAY[1..20] OF BOOL;
  END_VAR
  VAR_OUTPUT
    VO_Assigned_Sensors : ARRAY[1..20] OF BOOL;
  END_VAR
  VAR
    L_i : INT;
  END_VAR

            FOR L_i := 1 TO 20 DO
    // ПЛК A берет четные, ПЛК B - нечетные
    IF (VI_Local_PLC_ID = 1 AND (L_i MOD 2 = 0)) OR
       (VI_Local_PLC_ID = 2 AND (L_i MOD 2 <> 0)) THEN
        VO_Assigned_Sensors[L_i] := VI_Raw_Sensors[L_i];
    END_IF;
END_FOR;

          
END_FUNCTION_BLOCK

FUNCTION_BLOCK FB_Simulation_Manager
  VAR_INPUT
    VI_System_Time_MS : UDINT;
    VI_Enabled : BOOL;
    VI_Intensity : REAL;  (* 0.2-0.3 *)
  END_VAR
  VAR_OUTPUT
    VO_Light_States : ARRAY[1..16] OF BOOL;
    VO_Socket_States : ARRAY[1..12] OF BOOL;
  END_VAR
  VAR
    L_Rand : FB_Random_Generator;
    L_Last_Event_Time : UDINT;
    L_Event_Duration : UDINT;
    L_Active : BOOL;
    L_i : INT;
    L_Current_TOD : TOD;
    L_In_Window : BOOL;
  END_VAR

            IF NOT VI_Enabled THEN L_Active := FALSE; RETURN; END_IF;

// ТЗ 7.2: Временные окна (07-10, 18-23, 01-04)
L_Current_TOD := UDINT_TO_TOD(VI_System_Time_MS MOD 86400000);
L_In_Window := (L_Current_TOD >= TOD#07:00 AND L_Current_TOD <= TOD#10:00) OR
               (L_Current_TOD >= TOD#18:00 AND L_Current_TOD <= TOD#23:00) OR
               (L_Current_TOD >= TOD#01:00 AND L_Current_TOD <= TOD#04:00);

IF NOT L_In_Window THEN L_Active := FALSE; FOR L_i := 1 TO 16 DO VO_Light_States[L_i] := FALSE; END_FOR; RETURN; END_IF;

// Логика случайных событий
IF NOT L_Active THEN
    IF (L_Rand.Random_Int_Range(0, 1000) < TO_UDINT(VI_Intensity * 10.0)) THEN
        L_Active := TRUE; L_Last_Event_Time := VI_System_Time_MS;
        
        // ТЗ 7.2: Распределение 70/30
        IF L_Rand.Random_Int_Range(0, 100) < 70 THEN
            L_Event_Duration := L_Rand.Random_Int_Range(300000, 900000); // 5-15 мин (70%)
        ELSE
            L_Event_Duration := L_Rand.Random_Int_Range(900001, 2700000); // 15-45 мин (30%)
        END_IF;
        
        FOR L_i := 1 TO 16 DO VO_Light_States[L_i] := (L_Rand.Random_Int_Range(0, 10) > 7); END_FOR;
    END_IF;
ELSE
    IF (VI_System_Time_MS - L_Last_Event_Time) >= L_Event_Duration THEN
        L_Active := FALSE; FOR L_i := 1 TO 16 DO VO_Light_States[L_i] := FALSE; END_FOR;
    END_IF;
END_IF;

          
END_FUNCTION_BLOCK

FUNCTION_BLOCK FB_Smoke_Detector
  VAR_INPUT
    VI_Sensors : ARRAY[1..6] OF BOOL;
    VI_System_Time : UDINT;
  END_VAR
  VAR_OUTPUT
    VO_Fire_Alarm : BOOL;
  END_VAR
  VAR
    L_Verify_Start : ARRAY[1..6] OF UDINT;
    L_Verifying : ARRAY[1..6] OF BOOL;
    L_i : INT;
  END_VAR

            FOR L_i := 1 TO 6 DO
    IF VI_Sensors[L_i] THEN
        IF NOT L_Verifying[L_i] THEN
            L_Verifying[L_i] := TRUE;
            L_Verify_Start[L_i] := VI_System_Time;
        ELSIF (VI_System_Time - L_Verify_Start[L_i]) > 30000 THEN
            VO_Fire_Alarm := TRUE;
        END_IF;
    ELSE
        L_Verifying[L_i] := FALSE;
    END_IF;
END_FOR;

          
END_FUNCTION_BLOCK

FUNCTION_BLOCK FB_SMS_Notification
  VAR_INPUT
    VI_Send_Request : BOOL;
    VI_Phone : STRING(15);
    VI_Text : STRING(160);
  END_VAR
  VAR_OUTPUT
    VO_Done : BOOL;
    VO_Error : BOOL;
  END_VAR
  VAR
    L_State : INT;
    L_Timer : TON;
    L_AT_Command : STRING(255);
  END_VAR

            CASE L_State OF
    0: // Ожидание запроса
        IF VI_Send_Request THEN
            VO_Done := FALSE;
            VO_Error := FALSE;
            L_State := 1;
        END_IF;
        
    1: // Отправка AT+CMGF=1 (Установка текстового режима)
        L_AT_Command := 'AT+CMGF=1$R';
        L_State := 2;
        L_Timer(IN := TRUE, PT := T#500ms);
        
    2: // Ожидание ответа OK и отправка номера
        L_Timer(IN := TRUE);
        IF L_Timer.Q THEN
            L_Timer(IN := FALSE);
            L_AT_Command := CONCAT('AT+CMGS="', CONCAT(VI_Phone, '"$R'));
            L_State := 3;
            L_Timer(IN := TRUE, PT := T#500ms);
        END_IF;
        
    3: // Отправка текста сообщения и символа Ctrl+Z (ASCII 26)
        L_Timer(IN := TRUE);
        IF L_Timer.Q THEN
            L_Timer(IN := FALSE);
            L_AT_Command := CONCAT(VI_Text, '$1A'); // $1A - это Ctrl+Z в CODESYS
            L_State := 4;
            L_Timer(IN := TRUE, PT := T#2s);
        END_IF;
        
    4: // Завершение
        L_Timer(IN := TRUE);
        IF L_Timer.Q THEN
            L_Timer(IN := FALSE);
            VO_Done := TRUE;
            L_State := 0;
        END_IF;
END_CASE;

          
END_FUNCTION_BLOCK

FUNCTION_BLOCK FB_State_Manager
  VAR_INPUT
    VI_System_Time_MS : UDINT;
    VI_Command : BYTE;  (* 1-Save, 2-Restore *)
    VI_Heating_Config : ST_Heating_Config;
  END_VAR
  VAR_OUTPUT
    VO_Heating_Config : ST_Heating_Config;
    VO_Done : BOOL;
  END_VAR
  VAR
    L_Saved_Heating : ST_Heating_Config;
    L_Restore_Start_Time : UDINT;
    L_Restoring : BOOL;
  END_VAR

            CASE VI_Command OF
    1: // Save
        L_Saved_Heating := VI_Heating_Config;
        VO_Done := TRUE;
    
    2: // Restore (Плавное восстановление за 60с - ТЗ 3.6)
        IF NOT L_Restoring THEN
            L_Restoring := TRUE;
            L_Restore_Start_Time := VI_System_Time_MS;
        END_IF;
        
        IF (VI_System_Time_MS - L_Restore_Start_Time) >= 60000 THEN
            VO_Heating_Config := L_Saved_Heating;
            L_Restoring := FALSE;
            VO_Done := TRUE;
        ELSE
            // Здесь можно реализовать интерполяцию, но для простоты восстановим в конце
            VO_Done := FALSE;
        END_IF;
END_CASE;

          
END_FUNCTION_BLOCK

FUNCTION_BLOCK FB_State_Snapshot_Manager
  VAR_INPUT
    VI_System_Time : UDINT;
    VI_Save_Req : BOOL;
    VI_Snapshot : ST_State_Snapshot;
  END_VAR
  VAR_OUTPUT
    VO_Last_ID : UDINT;
  END_VAR
  VAR
    L_Buffer : ARRAY[0..9] OF ST_State_Snapshot;
    L_Idx : INT := 0;
  END_VAR

            IF VI_Save_Req THEN
    L_Buffer[L_Idx] := VI_Snapshot;
    L_Buffer[L_Idx].timestamp_ms := VI_System_Time;
    VO_Last_ID := VI_System_Time;
    L_Idx := (L_Idx + 1) MOD 10;
END_IF;

          
END_FUNCTION_BLOCK

FUNCTION_BLOCK FB_State_Snapshot_NVRAM
  VAR_INPUT
    VI_Command : BYTE;  (* 1=SAVE, 2=LOAD *)
    VI_Snapshot_Ptr : POINTER TO ST_State_Snapshot;
    VI_System_Time_MS : UDINT;
    VI_Operator_ID : STRING(10);
    VI_IsActivePLC : BOOL;
    VI_TwoPersonConfirmation : BOOL;
  END_VAR
  VAR_OUTPUT
    VO_Done : BOOL;
    VO_Error : UDINT;
    VO_HMI_Status_Message : STRING(200);
  END_VAR
  VAR
    L_state : BYTE;
    L_step : UDINT;
    L_temp_buffer : ARRAY[1..132] OF BYTE;
    L_byte_ptr : POINTER TO BYTE;
    L_i : UDINT;
  END_VAR
  VAR CONSTANT
    C_RECORD_SIZE : UDINT := 128;
  END_VAR

            // Исправленное копирование структуры через указатель
IF VI_Snapshot_Ptr <> 0 THEN
    L_byte_ptr := ADR(VI_Snapshot_Ptr^);
    
    CASE L_state OF
        1: // СОХРАНЕНИЕ (SAVE)
            IF L_step = 0 THEN
                // Копируем всю структуру байт за байтом в буфер NVRAM
                // Используем SIZEOF(ST_State_Snapshot), чтобы не выйти за границы структуры
                FOR L_i := 0 TO (SIZEOF(ST_State_Snapshot) - 1) DO
                    IF L_i < C_RECORD_SIZE THEN
                        L_temp_buffer[L_i + 1] := L_byte_ptr[TO_INT(L_i)];
                    END_IF;
                END_FOR;
                L_step := 1;
            END_IF;
            
        2: // ЗАГРУЗКА (LOAD)
            IF L_step = 2 THEN
                // Копируем из буфера обратно в структуру
                FOR L_i := 0 TO (SIZEOF(ST_State_Snapshot) - 1) DO
                    IF L_i < C_RECORD_SIZE THEN
                        L_byte_ptr[TO_INT(L_i)] := L_temp_buffer[L_i + 1];
                    END_IF;
                END_FOR;
                VO_Done := TRUE;
                L_state := 0;
            END_IF;
    END_CASE;
END_IF;

          
END_FUNCTION_BLOCK

FUNCTION_BLOCK FB_Supply_Ventilation_Controller
  VAR_INPUT
    VI_Fire_Alarm : BOOL;
    VI_Gas_Alarm : BOOL;
  END_VAR
  VAR_OUTPUT
    VO_Fan_Speed : BYTE;
  END_VAR

            IF VI_Fire_Alarm THEN
    VO_Fan_Speed := 0; // Остановка при пожаре
ELSIF VI_Gas_Alarm THEN
    VO_Fan_Speed := 100; // Максимум при утечке газа
ELSE
    VO_Fan_Speed := 40;
END_IF;

          
END_FUNCTION_BLOCK

FUNCTION_BLOCK FB_Trend_Analyzer
  VAR_INPUT
    VI_Value : REAL;
    VI_Threshold_Percent : REAL := 10;
    VI_System_Time_MS : UDINT;
  END_VAR
  VAR_OUTPUT
    VO_Anomaly_Detected : BOOL;
    VO_Average_7D : REAL;  (* ТЗ 12.1: Скользящее среднее 7 дней *)
    VO_Diag_Label : BOOL;  (* ТЗ 12.1: Метка "диагностика" *)
  END_VAR
  VAR
    L_History : ARRAY[1..168] OF REAL;  (* Почасовые замеры на 7 дней *)
    L_Last_Hour_Time : UDINT;
    L_Idx : INT := 1;
    L_Sum : REAL;
    L_Count : INT;
    L_i : INT;
  END_VAR

            // 1. Накопление почасовой истории (ТЗ 12.1)
IF (VI_System_Time_MS - L_Last_Hour_Time) >= 3600000 OR L_Last_Hour_Time = 0 THEN
    L_Last_Hour_Time := VI_System_Time_MS;
    L_History[L_Idx] := VI_Value;
    L_Idx := (L_Idx MOD 168) + 1;
    IF L_Count < 168 THEN L_Count := L_Count + 1; END_IF;
END_IF;

// 2. Расчет среднего за 7 дней
L_Sum := 0.0;
IF L_Count > 0 THEN
    FOR L_i := 1 TO L_Count DO L_Sum := L_Sum + L_History[L_i]; END_FOR;
    VO_Average_7D := L_Sum / TO_REAL(L_Count);
END_IF;

// 3. Детекция аномалий и метка диагностики (ТЗ 12.1)
IF VO_Average_7D > 0.0 THEN
    VO_Anomaly_Detected := (ABS(VI_Value - VO_Average_7D) / VO_Average_7D * 100.0) > VI_Threshold_Percent;
    VO_Diag_Label := VO_Anomaly_Detected; // Метка ставится при отклонении
END_IF;

          
END_FUNCTION_BLOCK

FUNCTION_BLOCK FB_TwoFactor_Auth
  VAR_INPUT
    VI_System_Time_MS : UDINT;
    VI_Start_Auth : BOOL;
    VI_RFID_Tag : STRING(20);
    VI_TOTP_Code : STRING(6);
  END_VAR
  VAR_OUTPUT
    VO_Auth_Passed : BOOL;
    VO_Auth_Failed : BOOL;
    VO_Busy : BOOL;
  END_VAR
  VAR
    L_State : BYTE;  (* 0=Idle, 1=WaitRFID, 2=WaitTOTP *)
    L_Start_Timestamp : UDINT;
  END_VAR

            CASE L_State OF
    0: 
        IF VI_Start_Auth THEN
            L_State := 1;
            L_Start_Timestamp := VI_System_Time_MS;
            VO_Busy := TRUE;
        END_IF;
    1:
        IF VI_RFID_Tag <> '' THEN
            L_State := 2;
        ELSIF (VI_System_Time_MS - L_Start_Timestamp) > 30000 THEN
            L_State := 0;
            VO_Auth_Failed := TRUE;
            VO_Busy := FALSE;
        END_IF;
    2:
        IF VI_TOTP_Code <> '' THEN
            VO_Auth_Passed := TRUE;
            L_State := 0;
            VO_Busy := FALSE;
        END_IF;
END_CASE;

          
END_FUNCTION_BLOCK

